(* IEC 61131-3 sources: elnaProjects/ElpcLogic/PomarKc7Unchanged/build_USO_ecl (part 7) *)

                                          StrAlg.inOpcCommandsDisabled:=FALSE;

  				cmd_for_Status := cmd;
  				source_for_Status := source;
  				command_error_for_Status := 0;
  	END_CASE;
  	resetCmdTimer(IN := false);
  	resetCmdTimerPriznak := TRUE;
  END_IF;
  lastCmd := cmd;

  resetCmdTimer(IN := resetCmdTimerPriznak, PT := T#5S);
  IF resetCmdTimer.Q THEN
  	resetCmdTimerPriznak := FALSE;
  	source_for_Status := 0;
  	cmd_for_Status := 0;
  	command_error_for_Status := 0;
  END_IF;

  StrAlg.Start:= puskOilSystem.startStatus
              OR nuOff.startStatus
              OR dPmgAi.startStatus
              OR dPmgDi.startStatus
              OR nuOn.startStatus
              OR noRezrv.startStatus
              OR BreakTest.startStatus
              OR testUnsuccessful.startStatus
              OR pnsOff.startStatus
              OR stopANU.startStatus
              OR nu1Off.startStatus
              OR nu2Off.startStatus;

  StrAlg.Error:=  puskOilSystem.errorStatus
              OR nuOff.errorStatus
              OR dPmgAi.errorStatus
              OR dPmgDi.errorStatus
              OR nuOn.errorStatus
              OR noRezrv.errorStatus
              OR BreakTest.errorStatus
              OR testUnsuccessful.errorStatus
              OR pnsOff.errorStatus
              OR stopANU.errorStatus
              OR nu1Off.errorStatus
              OR nu2Off.errorStatus;

  StrAlg.Top:=   puskOilSystem.topStatus
              OR nuOff.topStatus
              OR dPmgAi.topStatus
              OR dPmgDi.topStatus
              OR nuOn.topStatus
              OR noRezrv.topStatus
              OR BreakTest.topStatus
              OR testUnsuccessful.topStatus
              OR pnsOff.topStatus
              OR stopANU.topStatus
              OR nu1Off.topStatus
              OR nu2Off.topStatus;

  (*TODO: TYPE PROGRAM CODE HERE*)
  StrAlg.status :=  SHL(BYTE_TO_DWORD(source_for_Status), 29)
  			OR SHL(BYTE_TO_DWORD(cmd_for_Status), 26)
  			OR SHL(BYTE_TO_DWORD(command_error_for_Status), 23)
  			OR SHL(BOOL_TO_DWORD(StrAlg.OpcCommandsDisabled ), 21)
  			OR SHL(BOOL_TO_DWORD(StrAlg.hasError),4)
  			OR SHL(BOOL_TO_DWORD(StrAlg.CanRun),2)
  			OR SHL(BOOL_TO_DWORD(StrAlg.isEnded),1)
  			OR BOOL_TO_DWORD(StrAlg.isRuning);
END_FUNCTION_BLOCK

FUNCTION_BLOCK fb_ph_AIprotection
  VAR_IN_OUT
    StrAiP : struct_AiProtection;
  END_VAR
  VAR_INPUT
    act : TYPE_PhaseAlgoritmAction;
    PhaseNumber : UINT;
  END_VAR
  VAR_IN_OUT
    StrPh : struct_PhaseAlgoritm;
  END_VAR
  VAR
    CommandFault_Trig : R_TRIG;
    reset_Trig : R_TRIG;
    _statusDualInput : TYPE_statusDualInput;
  END_VAR

  IF StrPh.run AND NOT StrPh.start THEN
  	StrPh.start := TRUE;
  	StrPh.top := FALSE;
  	StrPh.error := FALSE;
            StrPh.run:=FALSE;

  	CASE act OF
  		(*PhaseAlgoritmAction.run*)    _run : runAiProtection(StrAiP); (*cmd_run*)
  		(*PhaseAlgoritmAction.reset*)_reset : resetAiProtection(StrAiP); (*cmd_reset*)
  	END_CASE;
  END_IF;

  IF StrPh.start AND NOT StrPh.top THEN
                      CommandFault_Trig(CLK := StrAiP.hasError);
                      IF CommandFault_Trig.Q THEN
  	          StrPh.error := TRUE;
                      END_IF;

  		CASE act OF
  		(*PhaseAlgoritmAction.run*)    _run:    StrPh.top:=StrAiP.isRunning;

  		(*PhaseAlgoritmAction.reset*) _reset:   StrPh.top := NOT StrAiP.isRunning;
  		END_CASE;

  END_IF;

  IF StrPh.top THEN
  StrPh.error := FALSE;
  END_IF;

  reset_Trig(CLK := StrPh.reset);
  IF reset_Trig.Q THEN
            StrPh.start := FALSE;
  	StrPh.error := FALSE;
  	StrPh.top := FALSE;
            StrPh.run:=FALSE;
            StrPh.reset:=FALSE;
  END_IF;

  StrPh.startStatus := SHL(BOOL_TO_DWORD(StrPh.start), PhaseNumber);
  StrPh.errorStatus := SHL(BOOL_TO_DWORD(StrPh.error), PhaseNumber);
  StrPh.topStatus := SHL(BOOL_TO_DWORD(StrPh.top), PhaseNumber);
END_FUNCTION_BLOCK

FUNCTION_BLOCK testPmsAlg
  VAR_IN_OUT
    StrAlg : struct_Alg;
    algContinue : struct_Question;
  END_VAR
  VAR
    pnsOn : struct_PhaseAlgoritm;
    PmsUp : struct_PhaseAlgoritm;
    runProtecrionAi : struct_PhaseAlgoritm;
    pnsOff : struct_PhaseAlgoritm;
    BreakTest : struct_PhaseAlgoritm;
    LowOilPS : struct_PhaseAlgoritm;
    LowOilAS : struct_PhaseAlgoritm;
    testUnsuccessful : struct_PhaseAlgoritm;
    fb_pnsOn : fb_ph_Switch;
    fb_PmsUp : fb_ph_WaitAnalogValue;
    fb_algContinue : fb_Question;
    fb_runProtecrionAi : fb_ph_AIprotection;
    fb_pnsOff : fb_ph_Switch;
    fb_BreakTest : fb_ph_Timer;
    fb_LowOilPS : fb_ph_CustomPhase;
    fb_LowOilAS : fb_ph_CustomPhase;
    fb_testUnsuccessful : fb_ph_CustomPhase;
    _sunpackerCommand : fb_sunpackerCommand;
    _DualStateImAction : TYPE_DualStateImAction;
    _Answers : TYPE_Answers;
    _statusDualInput : TYPE_statusDualInput;
    _StatusAi : TYPE_StatusAi;
    _PhaseAlgoritmAction : TYPE_PhaseAlgoritmAction;
    source : BYTE;
    cmd : BYTE;
    lastCmd : BYTE;
    source_for_Status : BYTE;
    cmd_for_Status : BYTE;
    command_error_for_Status : BYTE;
    resetCmdTimer : TON;
    resetCmdTimerPriznak : BOOL;
    onInit : BOOL;
    _resetQuestion : BOOL;
    waitReset : TON;
  END_VAR
  VAR_EXTERNAL
    IM : ImConfig;
    algoritms : AlgoritmsConfig;
    ai : AiConfig;
    AlgTimers : struct_AlgTimers;
    ModeGpa : TYPE_ModeGpa;
    algManager : struct_AlgoritmsManager;
    protections : ProtectionsConfig;
  END_VAR

  IF NOT onInit THEN

                     fb_pnsOn(phaseNumber:=0, act:=_on);
          algContinue.AnswerVariants:=_Answers.ANS_YES;
                     fb_PmsUp(phaseNumber:=1);
           fb_runProtecrionAi(phaseNumber:=3, act:=_run);
                    fb_pnsOff(phaseNumber:=4, act:=_off);
                 fb_BreakTest(phaseNumber:=5, delay:=T#120S);
                  fb_LowOilPS(phaseNumber:=6);
                  fb_LowOilAS(phaseNumber:=7);
          fb_testUnsuccessful(phaseNumber:=8);

  onInit:=TRUE;
  END_IF;

              fb_pnsOn(StrPh:=pnsOn, Im:=IM.pns);
        fb_algContinue(StrQ:=algContinue);
              fb_PmsUp(StrPh:=PmsUp, ai:=ai.P_masla_smazki_nizkoe, more:=ai.P_masla_smazki_nizkoe.LW);
    fb_runProtecrionAi(StrPh:=runProtecrionAi, StrAiP:=protections.P_masla_smazki_nizkoe_LA);
             fb_pnsOff(StrPh:=pnsOff, Im:=IM.pns);
          fb_BreakTest(StrPh:=BreakTest, timer:=AlgTimers.testPms_BreakTest);
           fb_LowOilPS(StrPh:=LowOilPS);
           fb_LowOilAS(StrPh:=LowOilAS);
   fb_testUnsuccessful(StrPh:=testUnsuccessful);

  StrAlg.CanRun := StrAlg.inCanRun;
  StrAlg.OpcCommandsDisabled := StrAlg.inOpcCommandsDisabled;

  IF StrAlg.isRuning THEN

      StrAlg.hasError := pnsOn.error OR pnsOff.error OR testUnsuccessful.error;

      IF pnsOn.top THEN
           runPhase(PmsUp);
      END_IF;

      IF PmsUp.top THEN
           runPhase(runProtecrionAi);
      END_IF;

      IF runProtecrionAi.top THEN
           IM.SingleSignals.P_oil_low.Disabled_Sig:=FALSE;
           ai.P_masla_smazki_nizkoe.Disabled_LA:=FALSE;
           ai.P_masla_smazki_nizkoe.Disabled_LW:=FALSE;
           ai.P_masla_smazki_srednee_posle_nasosov.Disabled_LW:=FALSE;
               IF NOT _resetQuestion THEN
                   askQuestion(algContinue);
                   _resetQuestion:=TRUE;
               END_IF;
      END_IF;

      IF algContinue.answer = _Answers.ANS_YES THEN

          runPhase(BreakTest);
          runPhase(pnsOff);
          runPhase(LowOilPS);
          runPhase(LowOilAS);
          resetQuestion(algContinue);

      END_IF;

      IF 	LowOilPS.start AND NOT LowOilPS.top THEN
  	LowOilPS.top:= ai.P_masla_smazki_nizkoe.interval = _statusAi.LW;
      END_IF;
      IF 	LowOilAS.start AND NOT LowOilAS.top THEN
  	LowOilAS.top:= ai.P_masla_smazki_nizkoe.interval = _statusAi.LA;
      END_IF;

      IF LowOilPS.top AND LowOilAS.top THEN
            resetPhase(BreakTest);
            waitReset(IN:=TRUE, PT:= T#3S);
      END_IF;

      IF BreakTest.top AND StrAlg.isEnded THEN
  	testUnsuccessful.error:=TRUE;
      END_IF;

      IF waitReset.Q THEN
          algManager.nMode:=ModeGpa.MODE_STOP;
          resetIfRunning(StrAlg);
      END_IF;

      StrAlg.isEnded:= LowOilPS.top AND LowOilAS.top;

  END_IF;

  StrAlg.CanRun := StrAlg.inCanRun;
  StrAlg.OpcCommandsDisabled := StrAlg.inOpcCommandsDisabled;

  (* ---- Если управление с ВУ заблокировано, то  передаем команду из алгоритма ---- *)
  IF StrAlg.inOpcCommandsDisabled THEN
  	StrAlg.inCommand := StrAlg.inCommand_Alg;
  ELSE (* иначе передаем команду с АРМа*)
  	StrAlg.inCommand := StrAlg.inCommand_ARM;
  END_IF;

  _sunpackerCommand(command := StrAlg.inCommand);
  	source := _sunpackerCommand.source;
  	cmd := _sunpackerCommand.cmd;

  IF cmd <> 0 AND lastCmd <> cmd AND (((NOT StrAlg.opcCommandsDisabled) AND source > 0) OR source = 0) then
  	CASE BYTE_TO_INT(cmd) OF
  		(*cmdRun*) 1: 	IF (StrAlg.CanRun) THEN
  					StrAlg.isRuning := TRUE;
  					StrAlg.isEnded := FALSE;
  					StrAlg.hasError := FALSE;
  					(*****************       OnRun       *****************)

                                                    algManager.nMode:=ModeGpa.MODE_TESTPMS;
                                                    resetAndDisable(alg:=algoritms.ppu);
                                                    runPhase(pnsOn);

  					cmd_for_Status := cmd;
  					source_for_Status := source;
  					command_error_for_Status := 0;
  				ELSE
  					StrAlg.isRuning := FALSE;
  					StrAlg.isEnded := FALSE;
  					StrAlg.hasError 	:= FALSE;

  					cmd_for_Status := 0;
  					source_for_Status := source;
  					command_error_for_Status := cmd;
  				END_IF;
  		(*cmdReset*) 2: 	StrAlg.isRuning := FALSE;
  				StrAlg.isEnded := FALSE;
  				StrAlg.hasError 	:= FALSE;

                                           (*****************       OnReset       *****************)
                                          waitReset(IN:=FALSE);
                                          _resetQuestion:=FALSE;
                                          ai.P_masla_smazki_nizkoe.Disabled_LA:=TRUE;
                                          ai.P_masla_smazki_nizkoe.Disabled_LW:=TRUE;
                                          ai.P_masla_smazki_srednee_posle_nasosov.Disabled_LW:=TRUE;
                                          IM.SingleSignals.P_oil_low.Disabled_Sig:=TRUE;
                                          resetAiProtection(protections.P_masla_smazki_nizkoe_LA);

                                          resetPhase(pnsOn);
                                          resetPhase(PmsUp);
                                          resetPhase(runProtecrionAi);
                                          resetPhase(pnsOff);
                                          resetPhase(BreakTest);
                                          resetPhase(LowOilPS);
                                          resetPhase(LowOilAS);
                                          resetPhase(testUnsuccessful);

                                          resetQuestion(algContinue);

                                          StrAlg.inOpcCommandsDisabled:=FALSE;

  				cmd_for_Status := cmd;
  				source_for_Status := source;
  				command_error_for_Status := 0;
  	END_CASE;
  	resetCmdTimer(IN := false);
  	resetCmdTimerPriznak := TRUE;
  END_IF;
  lastCmd := cmd;

  resetCmdTimer(IN := resetCmdTimerPriznak, PT := T#5S);
  IF resetCmdTimer.Q THEN
  	resetCmdTimerPriznak := FALSE;
  	source_for_Status := 0;
  	cmd_for_Status := 0;
  	command_error_for_Status := 0;
  END_IF;

  StrAlg.Start:= pnsOn.startStatus
              OR PmsUp.startStatus
              OR runProtecrionAi.startStatus
              OR pnsOff.startStatus
              OR BreakTest.startStatus
              OR LowOilPS.startStatus
              OR LowOilAS.startStatus
              OR testUnsuccessful.startStatus;

  StrAlg.Error:= pnsOn.errorStatus
              OR PmsUp.errorStatus
              OR runProtecrionAi.errorStatus
              OR pnsOff.errorStatus
              OR BreakTest.errorStatus
              OR LowOilPS.errorStatus
              OR LowOilAS.errorStatus
              OR testUnsuccessful.errorStatus;

  StrAlg.Top:=   pnsOn.topStatus
              OR PmsUp.topStatus
              OR runProtecrionAi.topStatus
              OR pnsOff.topStatus
              OR BreakTest.topStatus
              OR LowOilPS.topStatus
              OR LowOilAS.topStatus
              OR testUnsuccessful.topStatus;

  (*TODO: TYPE PROGRAM CODE HERE*)
  StrAlg.status :=  SHL(BYTE_TO_DWORD(source_for_Status), 29)
  			OR SHL(BYTE_TO_DWORD(cmd_for_Status), 26)
  			OR SHL(BYTE_TO_DWORD(command_error_for_Status), 23)
  			OR SHL(BOOL_TO_DWORD(StrAlg.OpcCommandsDisabled ), 21)
  			OR SHL(BOOL_TO_DWORD(StrAlg.hasError),4)
  			OR SHL(BOOL_TO_DWORD(StrAlg.CanRun),2)
  			OR SHL(BOOL_TO_DWORD(StrAlg.isEnded),1)
  			OR BOOL_TO_DWORD(StrAlg.isRuning);
END_FUNCTION_BLOCK

FUNCTION_BLOCK ApuskAlg
  VAR_IN_OUT
    StrAlg : struct_Alg;
  END_VAR
  VAR
    runOilsystem : struct_PhaseAlgoritm;
    runEngine : struct_PhaseAlgoritm;
    filling : struct_PhaseAlgoritm;
    fb_runOilsystem : fb_ph_algoritm;
    fb_runEngine : fb_ph_algoritm;
    fb_filling : fb_ph_algoritm;
    _sunpackerCommand : fb_sunpackerCommand;
    _PhaseAlgoritmAction : TYPE_PhaseAlgoritmAction;
    _statusDualInput : TYPE_statusDualInput;
    source : BYTE;
    cmd : BYTE;
    lastCmd : BYTE;
    source_for_Status : BYTE;
    cmd_for_Status : BYTE;
    command_error_for_Status : BYTE;
    resetCmdTimer : TON;
    resetCmdTimerPriznak : BOOL;
    onInit : BOOL;
    waitReset : TON;
  END_VAR
  VAR_EXTERNAL
    algoritms : AlgoritmsConfig;
    ModeGpa : TYPE_ModeGpa;
    algManager : struct_AlgoritmsManager;
    IM : ImConfig;
  END_VAR

  IF NOT onInit THEN

           fb_runOilsystem(phaseNumber:=0, act:=_run, waitCompletion:=TRUE);
              fb_runEngine(phaseNumber:=1, act:=_run, waitCompletion:=TRUE);
                fb_filling(phaseNumber:=2, act:=_run, waitCompletion:=TRUE);

  onInit:=TRUE;
  END_IF;

           fb_runOilsystem(StrPh:=runOilsystem, alg:=algoritms.puskOilSystem);
              fb_runEngine(StrPh:=runEngine, alg:=algoritms.engineRun);
                fb_filling(StrPh:=filling, alg:=algoritms.filling);

  StrAlg.CanRun := StrAlg.inCanRun;
  StrAlg.OpcCommandsDisabled := StrAlg.inOpcCommandsDisabled;

  IF StrAlg.isRuning THEN

      StrAlg.hasError := runOilsystem.error OR runEngine.error OR filling.error;

      IF runOilsystem.top THEN
           runPhase(runEngine);
      END_IF;

      IF runEngine.top THEN
           runPhase(filling);
      END_IF;

      IF filling.top THEN
            waitReset(IN:=TRUE, PT:= T#2S);
      END_IF;

      IF waitReset.Q THEN

          IF Im.kran6.onStatus = _statusDualInput.STATUS_On THEN
  	algManager.nMode:= ModeGpa.MODE_WORK_Ring;
          END_IF;
          IF Im.kran6.onStatus = _statusDualInput.STATUS_Off THEN
  	algManager.nMode:= ModeGpa.MODE_WORK_Line;
          END_IF;

          resetIfRunning(StrAlg);
      END_IF;

      StrAlg.isEnded:= filling.top;

  END_IF;

  StrAlg.CanRun := StrAlg.inCanRun;
  StrAlg.OpcCommandsDisabled := StrAlg.inOpcCommandsDisabled;

  (* ---- Если управление с ВУ заблокировано, то  передаем команду из алгоритма ---- *)
  IF StrAlg.inOpcCommandsDisabled THEN
  	StrAlg.inCommand := StrAlg.inCommand_Alg;
  ELSE (* иначе передаем команду с АРМа*)
  	StrAlg.inCommand := StrAlg.inCommand_ARM;
  END_IF;

  _sunpackerCommand(command := StrAlg.inCommand);
  	source := _sunpackerCommand.source;
  	cmd := _sunpackerCommand.cmd;

  IF cmd <> 0 AND lastCmd <> cmd AND (((NOT StrAlg.opcCommandsDisabled) AND source > 0) OR source = 0) then
  	CASE BYTE_TO_INT(cmd) OF
  		(*cmdRun*) 1: 	IF (StrAlg.CanRun) THEN
  					StrAlg.isRuning := TRUE;
  					StrAlg.isEnded := FALSE;
  					StrAlg.hasError := FALSE;
  					(*****************       OnRun       *****************)

                                                    algoritms.puskOilSystem.inCanRun:= TRUE	;
                                                    algoritms.filling.inCanRun:= TRUE	;
                                                    algoritms.engineRun.inCanRun:= TRUE	;

                                                    algManager.nMode:=ModeGpa.MODE_APUSK;
                                                    impulseSO(Im.SingleOutputs.VzvodBREO);
                                                    runPhase(runOilsystem);

  					cmd_for_Status := cmd;
  					source_for_Status := source;
  					command_error_for_Status := 0;
  				ELSE
  					StrAlg.isRuning := FALSE;
  					StrAlg.isEnded := FALSE;
  					StrAlg.hasError 	:= FALSE;

  					cmd_for_Status := 0;
  					source_for_Status := source;
  					command_error_for_Status := cmd;
  				END_IF;
  		(*cmdReset*) 2: 	StrAlg.isRuning := FALSE;
  				StrAlg.isEnded := FALSE;
  				StrAlg.hasError 	:= FALSE;

                                           (*****************       OnReset       *****************)
                                          waitReset(IN:=FALSE);
                                          StrAlg.inCanRun:=FALSE;

                                          resetPhase(runOilsystem);
                                          resetPhase(runEngine);
                                          resetPhase(filling);

                                          StrAlg.inOpcCommandsDisabled:=FALSE;

  				cmd_for_Status := cmd;
  				source_for_Status := source;
  				command_error_for_Status := 0;
  	END_CASE;
  	resetCmdTimer(IN := false);
  	resetCmdTimerPriznak := TRUE;
  END_IF;
  lastCmd := cmd;

  resetCmdTimer(IN := resetCmdTimerPriznak, PT := T#5S);
  IF resetCmdTimer.Q THEN
  	resetCmdTimerPriznak := FALSE;
  	source_for_Status := 0;
  	cmd_for_Status := 0;
  	command_error_for_Status := 0;
  END_IF;

  StrAlg.Start:= runOilsystem.startStatus
              OR runEngine.startStatus
              OR filling.startStatus;

  StrAlg.Error:= runOilsystem.errorStatus
              OR runEngine.errorStatus
              OR filling.errorStatus;

  StrAlg.Top:=   runOilsystem.topStatus
              OR runEngine.topStatus
              OR filling.topStatus;

  (*TODO: TYPE PROGRAM CODE HERE*)
  StrAlg.status :=  SHL(BYTE_TO_DWORD(source_for_Status), 29)
  			OR SHL(BYTE_TO_DWORD(cmd_for_Status), 26)
  			OR SHL(BYTE_TO_DWORD(command_error_for_Status), 23)
  			OR SHL(BOOL_TO_DWORD(StrAlg.OpcCommandsDisabled ), 21)
  			OR SHL(BOOL_TO_DWORD(StrAlg.hasError),4)
  			OR SHL(BOOL_TO_DWORD(StrAlg.CanRun),2)
  			OR SHL(BOOL_TO_DWORD(StrAlg.isEnded),1)
  			OR BOOL_TO_DWORD(StrAlg.isRuning);
END_FUNCTION_BLOCK

FUNCTION_BLOCK SemiAutoPuskAlg
  VAR_IN_OUT
    StrAlg : struct_Alg;
  END_VAR
  VAR
    runOilsystem : struct_PhaseAlgoritm;
    runEngine : struct_PhaseAlgoritm;
    filling : struct_PhaseAlgoritm;
  END_VAR
  VAR_IN_OUT
    cmdRun1ph : struct_Question;
    cmdRun2ph : struct_Question;
    cmdRun3ph : struct_Question;
  END_VAR
  VAR
    fb_runOilsystem : fb_ph_algoritm;
    fb_runEngine : fb_ph_algoritm;
    fb_filling : fb_ph_algoritm;
    fb_cmdRun1ph : fb_Question;
    fb_cmdRun2ph : fb_Question;
    fb_cmdRun3ph : fb_Question;
    _sunpackerCommand : fb_sunpackerCommand;
    _PhaseAlgoritmAction : TYPE_PhaseAlgoritmAction;
    _statusDualInput : TYPE_statusDualInput;
    _Answers : TYPE_Answers;
    source : BYTE;
    cmd : BYTE;
    lastCmd : BYTE;
    source_for_Status : BYTE;
    cmd_for_Status : BYTE;
    command_error_for_Status : BYTE;
    resetCmdTimer : TON;
    resetCmdTimerPriznak : BOOL;
    onInit : BOOL;
    waitReset : TON;
  END_VAR
  VAR_EXTERNAL
    algoritms : AlgoritmsConfig;
    ModeGpa : TYPE_ModeGpa;
    algManager : struct_AlgoritmsManager;
    IM : ImConfig;
  END_VAR

  IF NOT onInit THEN
                 cmdRun1ph.AnswerVariants:=_Answers.ANS_YES;
           fb_runOilsystem(phaseNumber:=0, act:=_run, waitCompletion:=TRUE);
                 cmdRun2ph.AnswerVariants:=_Answers.ANS_YES;
              fb_runEngine(phaseNumber:=1, act:=_run, waitCompletion:=TRUE);
                 cmdRun3ph.AnswerVariants:=_Answers.ANS_YES;
                fb_filling(phaseNumber:=2, act:=_run, waitCompletion:=TRUE);

  onInit:=TRUE;
  END_IF;
              fb_cmdRun1ph(StrQ:=cmdRun1ph);
           fb_runOilsystem(StrPh:=runOilsystem, alg:=algoritms.puskOilSystem);
              fb_cmdRun2ph(StrQ:=cmdRun2ph);
              fb_runEngine(StrPh:=runEngine, alg:=algoritms.engineRun);
              fb_cmdRun3ph(StrQ:=cmdRun3ph);
                fb_filling(StrPh:=filling, alg:=algoritms.filling);

  StrAlg.CanRun := StrAlg.inCanRun;
  StrAlg.OpcCommandsDisabled := StrAlg.inOpcCommandsDisabled;

  IF StrAlg.isRuning THEN

      StrAlg.hasError := runOilsystem.error OR runEngine.error OR filling.error;

      IF cmdRun1ph.answer = _Answers.ANS_YES THEN
  	runPhase(runOilsystem);
            resetQuestion(cmdRun1ph);
      END_IF;

      IF runOilsystem.top AND NOT runEngine.start THEN
           askQuestion(cmdRun2ph);
      END_IF;

      IF cmdRun2ph.answer = _Answers.ANS_YES THEN
           runPhase(runEngine);
           resetQuestion(cmdRun2ph);
      END_IF;

      IF runEngine.top AND NOT filling.start THEN
           askQuestion(cmdRun3ph);
      END_IF;

      IF cmdRun3ph.answer = _Answers.ANS_YES THEN
           runPhase(filling);
           resetQuestion(cmdRun3ph);
      END_IF;

      IF filling.top THEN
            waitReset(IN:=TRUE, PT:= T#2S);
      END_IF;

      IF waitReset.Q THEN

          IF Im.kran6.onStatus = _statusDualInput.STATUS_On THEN
  	algManager.nMode:= ModeGpa.MODE_WORK_Ring;
          END_IF;
          IF Im.kran6.onStatus = _statusDualInput.STATUS_Off THEN
  	algManager.nMode:= ModeGpa.MODE_WORK_Line;
          END_IF;

          resetIfRunning(StrAlg);
      END_IF;

      StrAlg.isEnded:= filling.top;

  END_IF;

  StrAlg.CanRun := StrAlg.inCanRun;
  StrAlg.OpcCommandsDisabled := StrAlg.inOpcCommandsDisabled;

  (* ---- Если управление с ВУ заблокировано, то  передаем команду из алгоритма ---- *)
  IF StrAlg.inOpcCommandsDisabled THEN
  	StrAlg.inCommand := StrAlg.inCommand_Alg;
  ELSE (* иначе передаем команду с АРМа*)
  	StrAlg.inCommand := StrAlg.inCommand_ARM;
  END_IF;

  _sunpackerCommand(command := StrAlg.inCommand);
  	source := _sunpackerCommand.source;
  	cmd := _sunpackerCommand.cmd;

  IF cmd <> 0 AND lastCmd <> cmd AND (((NOT StrAlg.opcCommandsDisabled) AND source > 0) OR source = 0) then
  	CASE BYTE_TO_INT(cmd) OF
  		(*cmdRun*) 1: 	IF (StrAlg.CanRun) THEN
  					StrAlg.isRuning := TRUE;
  					StrAlg.isEnded := FALSE;
  					StrAlg.hasError := FALSE;
  					(*****************       OnRun       *****************)

                                                    algoritms.puskOilSystem.inCanRun:= TRUE	;
                                                    algoritms.filling.inCanRun:= TRUE	;
                                                    algoritms.engineRun.inCanRun:= TRUE	;

                                                    algManager.nMode:=ModeGpa.MODE_MPUSK;
                                                    impulseSO(Im.SingleOutputs.VzvodBREO);
                                                    askQuestion(cmdRun1ph);

  					cmd_for_Status := cmd;
  					source_for_Status := source;
  					command_error_for_Status := 0;
  				ELSE
  					StrAlg.isRuning := FALSE;
  					StrAlg.isEnded := FALSE;
  					StrAlg.hasError 	:= FALSE;

  					cmd_for_Status := 0;
  					source_for_Status := source;
  					command_error_for_Status := cmd;
  				END_IF;
  		(*cmdReset*) 2: 	StrAlg.isRuning := FALSE;
  				StrAlg.isEnded := FALSE;
  				StrAlg.hasError 	:= FALSE;

                                           (*****************       OnReset       *****************)
                                          waitReset(IN:=FALSE);
                                          StrAlg.inCanRun:=FALSE;

                                          resetPhase(runOilsystem);
                                          resetPhase(runEngine);
                                          resetPhase(filling);

                                          resetQuestion(cmdRun1ph);
                                          resetQuestion(cmdRun2ph);
                                          resetQuestion(cmdRun3ph);

                                          StrAlg.inOpcCommandsDisabled:=FALSE;

  				cmd_for_Status := cmd;
  				source_for_Status := source;
  				command_error_for_Status := 0;
  	END_CASE;
  	resetCmdTimer(IN := false);
  	resetCmdTimerPriznak := TRUE;
  END_IF;
  lastCmd := cmd;

  resetCmdTimer(IN := resetCmdTimerPriznak, PT := T#5S);
  IF resetCmdTimer.Q THEN
  	resetCmdTimerPriznak := FALSE;
  	source_for_Status := 0;
  	cmd_for_Status := 0;
  	command_error_for_Status := 0;
  END_IF;

  StrAlg.Start:= runOilsystem.startStatus
              OR runEngine.startStatus
              OR filling.startStatus;

  StrAlg.Error:= runOilsystem.errorStatus
              OR runEngine.errorStatus
              OR filling.errorStatus;

  StrAlg.Top:=   runOilsystem.topStatus
              OR runEngine.topStatus
              OR filling.topStatus;

  (*TODO: TYPE PROGRAM CODE HERE*)
  StrAlg.status :=  SHL(BYTE_TO_DWORD(source_for_Status), 29)
  			OR SHL(BYTE_TO_DWORD(cmd_for_Status), 26)
  			OR SHL(BYTE_TO_DWORD(command_error_for_Status), 23)
  			OR SHL(BOOL_TO_DWORD(StrAlg.OpcCommandsDisabled ), 21)
  			OR SHL(BOOL_TO_DWORD(StrAlg.hasError),4)
  			OR SHL(BOOL_TO_DWORD(StrAlg.CanRun),2)
  			OR SHL(BOOL_TO_DWORD(StrAlg.isEnded),1)
  			OR BOOL_TO_DWORD(StrAlg.isRuning);
END_FUNCTION_BLOCK

FUNCTION_BLOCK proc_algoritms
  VAR
    fb_RemontAlg : RemontAlg;
    fb_TestProtectionAlg : TestProtectionAlg;
    fb_TestImAlg : TestImAlg;
    fb_AutoTen : fb_AutoTenAlg;
    fb_AutoPns : fb_AutoPnsAlg;
    fb_AutoAvom : fb_AutoAvomAlg;
    fb_vibegPNS : fb_vibegPNSAlg;
    fb_AutoNU : fb_AutoNUAlg;
    fb_puskOilSystem : fb_puskOilSystemAlg;
    fb_AntiPompag : fb_AntiPompagAlg;
    fb_NOAlg : NOAlg;
    fb_AOAlg : AOAlg;
    fb_ppuALG : ppuAlg;
    fb_fillingAlg : fillingAlg;
    fb_engineRunAlg : engineRunAlg;
    fb_puskKalg : puskKalg;
    fb_puskValg : puskValg;
    fb_testdPmgAlg : testdPmgAlg;
    fb_testPmsAlg : testPmsAlg;
    fb_ApuskAlg : ApuskAlg;
    fb_SemiAutoPuskAlg : SemiAutoPuskAlg;
  END_VAR
  VAR_EXTERNAL
    algoritms : AlgoritmsConfig;
    AlgQuestions : AlgoritmsQuestions;
    ai : AiConfig;
    IM : ImConfig;
    AlgTimers : struct_AlgTimers;
  END_VAR

  fb_RemontAlg(StrAlg:=algoritms.Remont);

  fb_TestProtectionAlg(StrAlg:=algoritms.TestProtection);

  fb_TestImAlg(StrAlg:=algoritms.testIm);

  fb_AutoTen(StrAlg:= algoritms.AutoTen,
  T_masla:= ai.T_masla_v_maslobake,
  Uroven_masla:= ai.Uroven_masla_v_maslobake,
  offTemperature:= Im.AutoTen_offTemperature,
  TEN:= Im.Ten,
  PNS:= Im.pns);

  fb_AutoPns(StrAlg:= algoritms.AutoPns,
  Poil:= ai.P_masla_smazki_nizkoe,
  Ust_Run:= Im.AutoPns_UstRun,
  Ust_Stop:= Im.AutoPns_UstStop,
  Nasos:= Im.pns,
  diPlow:= Im.SingleSignals.P_oil_low);

  fb_AutoAvom(StrAlg:= algoritms.AutoAvom,
  im1:= Im.v1_Avom,
  im2:= Im.v2_Avom,
  on1Temperature:= Im.AutoAvom_onTemp1,
  on2Temperature:= Im.AutoAvom_onTemp2,
  hystereses:= Im.AutoAvom_hysteresis,
  ai:= ai.T_masla_posle_AVOM);

  fb_vibegPNS(StrAlg:=algoritms.vibegPNS,
  algContinue:=AlgQuestions.vibegPNS_algContinue
  );

  fb_AutoNU(StrAlg:=algoritms.autoNu,
  nu1:=Im.nu1,
  nu2:=Im.nu2,
  Ust_Swap:= Im.AutoNU_Ust_Swap,
  mainNU:= Im.AutoNU_mainNU,
  dPoil:=ai.dPmaslo_gaz,
  Lowdp_di:=Im.SingleSignals.dP_oilgaz_low
  );

  fb_puskOilSystem(StrAlg:=algoritms.puskOilSystem);

  fb_AntiPompag(StrAlg:=algoritms.AntiPompag,
  Rashod:= ai.Rashod,
  Zapas:= ai.Zapas,
  P_gasIn:=ai.P_gaza_na_vkhode_nagnetatelia,
  T_gasIn:=ai.T_gaz_in_nagnetatelia,
  dP_konf:=ai.dP_gaza_na_konfuzore_nagnetatelia,
  Kran6:= im.Kran6,
  UgolVNA:= im.AntiPompag_UgolVNA,
  K:=im.AntiPompag_K,
  A:=im.AntiPompag_A,
  y0:=im.AntiPompag_y0);

  fb_NOAlg(StrAlg:=algoritms.no);

  fb_AOAlg(StrAlg:=algoritms.ao);

  fb_ppuAlg(StrAlg:=algoritms.ppu);

  fb_fillingAlg(StrAlg:=algoritms.filling);

  fb_engineRunAlg(StrAlg:=algoritms.engineRun);

  fb_puskKalg(StrAlg:=algoritms.puskK,
  questionFilling:=AlgQuestions.puskK_questionFilling,
   questionUnload:=AlgQuestions.puskK_questionUnload
  );

  fb_puskValg(StrAlg:=algoritms.puskV,
   questionEngine:=AlgQuestions.puskV_questionEngine,
    questionMVoff:=AlgQuestions.puskV_questionMVoff
  );

  fb_testdPmgAlg(StrAlg:=algoritms.testdPmg,
   algContinue:=AlgQuestions.testdPmg_algContinue
  );

  fb_testPmsAlg(StrAlg:=algoritms.testPms,
   algContinue:=AlgQuestions.testPms_algContinue
  );

  fb_ApuskAlg(StrAlg:=algoritms.Apusk);

  fb_SemiAutoPuskAlg(StrAlg:=algoritms.SemiAutoPusk,
   cmdRun1ph:=AlgQuestions.SemiAutoPusk_cmdRun1ph,
   cmdRun2ph:=AlgQuestions.SemiAutoPusk_cmdRun2ph,
   cmdRun3ph:=AlgQuestions.SemiAutoPusk_cmdRun3ph
  );
END_FUNCTION_BLOCK

FUNCTION anyProtectionSignaling : BOOL
  VAR_INPUT
    protections : ProtectionsConfig;
  END_VAR

  anyProtectionSignaling:=
  protections.T_perednego_opornogo_podshipnika_dvigatelia_t1_HA.Signaling OR
  protections.T_zadnego_opornogo_podshipnika_dvigatelia_t2_HA.Signaling OR
  protections.T_podshipnika_reduktora_t1_HA.Signaling OR
  protections.T_podshipnika_reduktora_t2_HA.Signaling OR
  protections.T_podshipnika_reduktora_t3_HA.Signaling OR
  protections.T_podshipnika_reduktora_t4_HA.Signaling OR
  protections.T_opornogo_podshipnika_nagnetatelia_t1_HA.Signaling OR
  protections.T_opornogo_podshipnika_nagnetatelia_t2_HA.Signaling OR
  protections.T_opornogo_podshipnika_nagnetatelia_t3_HA.Signaling OR
  protections.T_opornoupornogo_podshipnika_nagnetatelia_t4_HA.Signaling OR
  protections.T_gaza_na_vykhode_nagnetatelia_HA.Signaling OR
  protections.dP_maslogaz_LA.Signaling OR
  protections.P_masla_smazki_nizkoe_LA.Signaling OR
  protections.Vibratciia_STD_t1_HA.Signaling OR
  protections.Vibratciia_STD_t2_HA.Signaling OR
  protections.Vibratciia_rotora_nagnetatelia_t1_HA.Signaling OR
  protections.Vibratciia_rotora_nagnetatelia_t2_HA.Signaling OR
  protections.Vibratciia_rotora_nagnetatelia_t3_HA.Signaling OR
  protections.Vibratciia_rotora_nagnetatelia_t4_HA.Signaling OR
  protections.Osevoi_sdvig_rotora_nagnetatelia_HA.Signaling OR
  protections.Uroven_masla_v_maslobake_LA.Signaling OR
  protections.OsevojSdvigPravyjDi.Signaling OR
  protections.OsevojSdvigLevyjDi.Signaling OR
  protections.dP_masloGaz_LowDI.Signaling OR
  protections.DavlenieMaslaSmazkiDi.Signaling OR
  protections.mvOff.Signaling OR
  protections.NeispravnostVozbuzhdenijaDi.Signaling OR
  protections.AO_KC.Signaling OR
  protections.AO_PRU.Signaling OR
  protections.AO_SHU.Signaling OR
  protections.Srab_BEAO.Signaling OR
  protections.EAO_PRU.Signaling OR
  protections.BEAO_knSHU.Signaling OR
  protections.Kran1sdvig.Signaling OR
  protections.Kran2sdvig.Signaling;
END_FUNCTION

FUNCTION anyAnalogsPs : BOOL
  VAR_INPUT
    ai : AiConfig;
  END_VAR
  VAR
    statusAi : TYPE_StatusAi;
  END_VAR

  anyAnalogsPs:=
  ai.T_masla_v_maslobake.interval= statusAi.HW OR
  ai.T_masla_v_maslobake.interval= statusAi.LW OR
  ai.T_perednego_opornogo_podshipnika_dvigatelia_t1.interval= statusAi.HW OR
  ai.T_zadnego_opornogo_podshipnika_dvigatelia_t2.interval= statusAi.HW OR
  ai.T_podshipnika_reduktora_t1.interval= statusAi.HW OR
  ai.T_podshipnika_reduktora_t2.interval= statusAi.HW OR
  ai.T_podshipnika_reduktora_t3.interval= statusAi.HW OR
  ai.T_podshipnika_reduktora_t4.interval= statusAi.HW OR
  ai.T_opornogo_podshipnika_nagnetatelia_t1.interval= statusAi.HW OR
  ai.T_opornogo_podshipnika_nagnetatelia_t2.interval= statusAi.HW OR
  ai.T_opornogo_podshipnika_nagnetatelia_t3.interval= statusAi.HW OR
  ai.T_oporno_upornogo_podshipnika_nagnetatelia_t4.interval= statusAi.HW OR
  ai.T_gaz_out_nagnetatelia.interval= statusAi.HW OR
  ai.dPmaslo_gaz.interval= statusAi.LW OR
  ai.P_masla_smazki_nizkoe.interval= statusAi.LW OR
  ai.P_masla_smazki_srednee_posle_nasosov.interval= statusAi.LW OR
  ai.Vibratciia_STD_t1.interval= statusAi.HW OR
  ai.Vibratciia_STD_t2.interval= statusAi.HW OR
  ai.Vibratciia_rotora_nagnetatelia_t1.interval= statusAi.HW OR
  ai.Vibratciia_rotora_nagnetatelia_t2.interval= statusAi.HW OR
  ai.Vibratciia_rotora_nagnetatelia_t3.interval= statusAi.HW OR
  ai.Vibratciia_rotora_nagnetatelia_t4.interval= statusAi.HW OR
  ai.Osevoi_sdvig_rotora_nagnetatelia.interval= statusAi.HW OR
  ai.Osevoi_sdvig_rotora_nagnetatelia.interval= statusAi.LW OR
  ai.Uroven_masla_v_maslobake.interval= statusAi.HW OR
  ai.Uroven_masla_v_maslobake.interval= statusAi.LW OR
  ai.T_vnytri_shkafa.interval= statusAi.HW OR
  ai.T_vnytri_shkafa.interval= statusAi.LW OR
  ai.VoltageSHU_osnovnoi_vvod.interval= statusAi.HW OR
  ai.VoltageSHU_osnovnoi_vvod.interval= statusAi.LW OR
  ai.VoltageSHU_rezervnyi_vvod.interval= statusAi.HW OR
  ai.VoltageSHU_rezervnyi_vvod.interval= statusAi.LW;
END_FUNCTION

FUNCTION anyDiscretPS : BOOL
  VAR_INPUT
    im : ImConfig;
  END_VAR

  anyDiscretPS:=
      Im.SingleSignals.KZ_10kv.Q                     OR
      Im.SingleSignals.Vozb_ProboiVentila.Q	 OR
      Im.SingleSignals.Vozb_AsinchHod.Q	           OR
      Im.SingleSignals.NS_ForsingVozbugdenia.Q       OR
      Im.SingleSignals.Vozb_AutoUprVozbuditela_off.Q OR
      Im.SingleSignals.Vozb_KontaktorON.Q;
END_FUNCTION

FUNCTION UnBlockAllProtections : BOOL
  VAR_IN_OUT
    protections : ProtectionsConfig;
  END_VAR

  protections.T_perednego_opornogo_podshipnika_dvigatelia_t1_HA.inOpcCommandsDisabled:=FALSE;
  protections.T_zadnego_opornogo_podshipnika_dvigatelia_t2_HA.inOpcCommandsDisabled:=FALSE;
  protections.T_podshipnika_reduktora_t1_HA.inOpcCommandsDisabled:=FALSE;
  protections.T_podshipnika_reduktora_t2_HA.inOpcCommandsDisabled:=FALSE;
  protections.T_podshipnika_reduktora_t3_HA.inOpcCommandsDisabled:=FALSE;
  protections.T_podshipnika_reduktora_t4_HA.inOpcCommandsDisabled:=FALSE;
  protections.T_opornogo_podshipnika_nagnetatelia_t1_HA.inOpcCommandsDisabled:=FALSE;
  protections.T_opornogo_podshipnika_nagnetatelia_t2_HA.inOpcCommandsDisabled:=FALSE;
  protections.T_opornogo_podshipnika_nagnetatelia_t3_HA.inOpcCommandsDisabled:=FALSE;
  protections.T_opornoupornogo_podshipnika_nagnetatelia_t4_HA.inOpcCommandsDisabled:=FALSE;
  protections.T_gaza_na_vykhode_nagnetatelia_HA.inOpcCommandsDisabled:=FALSE;
  protections.dP_maslogaz_LA.inOpcCommandsDisabled:=FALSE;
  protections.P_masla_smazki_nizkoe_LA.inOpcCommandsDisabled:=FALSE;
  protections.Vibratciia_STD_t1_HA.inOpcCommandsDisabled:=FALSE;
  protections.Vibratciia_STD_t2_HA.inOpcCommandsDisabled:=FALSE;
  protections.Vibratciia_rotora_nagnetatelia_t1_HA.inOpcCommandsDisabled:=FALSE;
  protections.Vibratciia_rotora_nagnetatelia_t2_HA.inOpcCommandsDisabled:=FALSE;
  protections.Vibratciia_rotora_nagnetatelia_t3_HA.inOpcCommandsDisabled:=FALSE;
  protections.Vibratciia_rotora_nagnetatelia_t4_HA.inOpcCommandsDisabled:=FALSE;
  protections.Osevoi_sdvig_rotora_nagnetatelia_HA.inOpcCommandsDisabled:=FALSE;
  protections.Uroven_masla_v_maslobake_LA.inOpcCommandsDisabled:=FALSE;
  protections.OsevojSdvigPravyjDi.inOpcCommandsDisabled:=FALSE;
  protections.OsevojSdvigLevyjDi.inOpcCommandsDisabled:=FALSE;
  protections.dP_masloGaz_LowDI.inOpcCommandsDisabled:=FALSE;
  protections.DavlenieMaslaSmazkiDi.inOpcCommandsDisabled:=FALSE;
  protections.mvOff.inOpcCommandsDisabled:=FALSE;
  protections.NeispravnostVozbuzhdenijaDi.inOpcCommandsDisabled:=FALSE;
  protections.AO_KC.inOpcCommandsDisabled:=FALSE;
  protections.AO_PRU.inOpcCommandsDisabled:=FALSE;
  protections.AO_SHU.inOpcCommandsDisabled:=FALSE;
  protections.Srab_BEAO.inOpcCommandsDisabled:=FALSE;
  protections.EAO_PRU.inOpcCommandsDisabled:=FALSE;
  protections.BEAO_knSHU.inOpcCommandsDisabled:=FALSE;
  protections.Kran1sdvig.inOpcCommandsDisabled:=FALSE;
  protections.Kran2sdvig.inOpcCommandsDisabled:=FALSE;
END_FUNCTION

FUNCTION_BLOCK fb_AlgoritmsManager
  VAR_IN_OUT
    str_AM : struct_AlgoritmsManager;
  END_VAR
  VAR
    onInit : BOOL;
  END_VAR
  VAR_EXTERNAL
    ai : AiConfig;
  END_VAR
  VAR
    EoTrig : R_TRIG;
    EoFTrig : F_TRIG;
    PsLampTrig : R_TRIG;
    PsLampFTrig : F_TRIG;
    Ring : R_TRIG;
    Line : R_TRIG;
    statusDualInput : TYPE_statusDualInput;
  END_VAR
  VAR_EXTERNAL
    IM : ImConfig;
    protections : ProtectionsConfig;
    algoritms : AlgoritmsConfig;
    ModeGpa : TYPE_ModeGpa;
  END_VAR

  IF NOT onInit THEN
            DisableAiLimits(ai);
            IM.SingleSignals.P_oil_low.Disabled_Sig:=TRUE;
            IM.SingleSignals.dP_oilgaz_low.Disabled_Sig:=TRUE;
            str_AM.nMode:=ModeGpa.MODE_STOP;
            BlockAllIM(IM);
            runIfNotRunning(algoritms.AutoTen);
  onInit:=TRUE;
  END_IF;

  str_AM.DiscretPS:=anyDiscretPS(IM);
  str_AM.AnalogsPs:=anyAnalogsPs(ai);
  str_AM.ProtectionSignaling:=anyProtectionSignaling(protections);

  EoTrig(CLK := IM.SingleSignals.BEO_Srabat.Q);
  IF EoTrig.Q THEN
  	stopPusk(algoritms);
  	resetAndDisable(algoritms.Remont);
  	resetAndDisable(algoritms.no);
  	resetAndDisable(algoritms.ao);
  	str_AM.nMode:=ModeGpa.MODE_EO;
  END_IF;
  EoFTrig(CLK := IM.SingleSignals.BEO_Srabat.Q);
  IF EoFTrig.Q THEN
  	str_AM.nMode:=ModeGpa.MODE_STOP;
  	runIfNotRunning(algoritms.ao);
  END_IF;

  IF (str_AM.ProtectionSignaling OR Im.SingleSignals.AO_KC.Q OR Im.SingleSignals.AOGPA_knopkaSHU.Q OR Im.SingleSignals.AOGPA_PRU.Q )
  	AND NOT((str_AM.mode=ModeGpa.MODE_AO) OR (str_AM.mode=ModeGpa.MODE_EO) OR IM.SingleOutputs.IndikicijaAS_fonar.Q
            OR (str_AM.mode=ModeGpa.MODE_TESTAZ) OR (str_AM.mode=ModeGpa.MODE_TESTDPMG) OR (str_AM.mode=ModeGpa.MODE_REMONT) OR
            (str_AM.mode=ModeGpa.MODE_TESTPMS))THEN
  		runIfNotRunning(algoritms.ao);
  	str_AM.nMode:=ModeGpa.MODE_AO;
  END_IF;

  IF Im.SingleSignals.NOGPA_knopkaSHU.Q  AND algoritms.no.CanRun THEN
  	runIfNotRunning(algoritms.no);
            str_AM.nMode:=ModeGpa.MODE_NO;
  END_IF;

  PsLampTrig(CLK := str_AM.DiscretPS OR str_AM.AnalogsPs);
  IF PsLampTrig.Q THEN
            runIfNotRunningSO(IM.SingleOutputs.IndikicijaPS_fonar);
  END_IF;
  PsLampFTrig(CLK := str_AM.DiscretPS OR str_AM.AnalogsPs);
  IF PsLampFTrig.Q THEN
            resetIfRunningSO(IM.SingleOutputs.IndikicijaPS_fonar);
  END_IF;

  IF str_AM.mode = ModeGpa.MODE_WORK_Line OR str_AM.mode = ModeGpa.MODE_WORK_Ring  THEN

  	Ring(CLK:=Im.kran6.onStatus=statusDualInput.STATUS_On);
  	Line(CLK:=Im.kran6.onStatus=statusDualInput.STATUS_Off);

  	IF Ring.Q AND str_AM.mode = ModeGpa.MODE_WORK_Line THEN
  		str_AM.nMode:=ModeGpa.MODE_WORK_Ring;
  	END_IF;
  	IF Line.Q AND str_AM.mode = ModeGpa.MODE_WORK_Ring THEN
  		str_AM.nMode:=ModeGpa.MODE_WORK_Line;
  	END_IF;

  END_IF;

  IF str_AM.mode = ModeGpa.MODE_WORK_Line THEN
            runIfNotRunning(alg:=algoritms.AntiPompag);
  	ELSE
            resetAndDisable(alg:=algoritms.AntiPompag);
  END_IF;

  IF str_AM.nMode<>str_AM.mode THEN
  	str_AM.mode:=str_AM.nMode;
  	CASE str_AM.mode OF
  	(*ModeGpa.MODE_REMONT*)1:
  		stopPusk(algoritms);
  		resetAndDisable(alg:=algoritms.no);
  		resetAndDisable(alg:=algoritms.ao);
  		resetAndDisable(alg:=algoritms.TestProtection);
                      resetAndDisable(alg:=algoritms.testIm);

  	(*ModeGpa.MODE_TESTAZ*)16:
  		stopPusk(algoritms);
  		resetAndDisable(alg:=algoritms.ao);
  		resetAndDisable(alg:=algoritms.no);
                      resetAndDisable(alg:=algoritms.Remont);
                      resetAndDisable(alg:=algoritms.testIm);

            (*ModeGpa.MODE_TESTIM*)15:
                      stopPusk(algoritms);
                      resetAndDisable(alg:=algoritms.Remont);
                      resetAndDisable(alg:=algoritms.TestProtection);

  	(*ModeGpa.MODE_EO*)14:
  		stopPusk(algoritms);
  		resetAndDisable(alg:=algoritms.no);
  		resetAndDisable(alg:=algoritms.ao);
  		resetAndDisable(alg:=algoritms.Remont);
                      resetAndDisable(alg:=algoritms.testIm);
                      resetAndDisable(alg:=algoritms.TestProtection);
  	(*ModeGpa.MODE_AO*)13:
  		(*//stopPusk();*)
  		resetAndDisable(alg:=algoritms.no);
  		resetAndDisable(alg:=algoritms.Remont);
                      resetAndDisable(alg:=algoritms.testIm);
                      resetAndDisable(alg:=algoritms.TestProtection);
                      algoritms.VibegPNS.inCanRun:=TRUE;
  	(*ModeGpa.MODE_NO*)12:
  		stopPusk(algoritms);
                      resetAndDisable(alg:=algoritms.testIm);
                      resetAndDisable(alg:=algoritms.Remont);
                      resetAndDisable(alg:=algoritms.TestProtection);
                      algoritms.VibegPNS.inCanRun:=TRUE;
  		algoritms.ao.inCanRun:=TRUE;
  	(*ModeGpa.MODE_APUSK*)8:
  		resetAndDisable(alg:=algoritms.SemiAutoPusk);
  		resetAndDisable(alg:=algoritms.puskV);
  		resetAndDisable(alg:=algoritms.puskK);
  		resetAndDisable(alg:=algoritms.testdPmg);
  		resetAndDisable(alg:=algoritms.testPms);
  		(*resetAndDisable(alg:=algoritms.testIm);
                      resetAndDisable(alg:=algoritms.TestProtection);
                      resetAndDisable(alg:=algoritms.Remont);*)
  		resetAndDisable(alg:=algoritms.ppu);
  		algoritms.no.inCanRun:=TRUE;
  		algoritms.ao.inCanRun:=TRUE;

  	(*ModeGpa.MODE_MPUSK*)9:
  		resetAndDisable(alg:=algoritms.Apusk);
  		resetAndDisable(alg:=algoritms.puskV);
  		resetAndDisable(alg:=algoritms.puskK);
  		resetAndDisable(alg:=algoritms.testdPmg);
  		resetAndDisable(alg:=algoritms.testPms);
  		(*resetAndDisable(alg:=algoritms.testIm);
                      resetAndDisable(alg:=algoritms.TestProtection);
                      resetAndDisable(alg:=algoritms.Remont);	*)
  		resetAndDisable(alg:=algoritms.ppu);
  		algoritms.no.inCanRun:=TRUE;
                      algoritms.no.inOpcCommandsDisabled:=FALSE;
  		algoritms.ao.inCanRun:=TRUE;
                      algoritms.ao.inOpcCommandsDisabled:=FALSE;

  	(*ModeGpa.MODE_PUSKK*)5:
                      resetAndDisable(alg:=algoritms.ppu);
  		resetAndDisable(alg:=algoritms.Apusk);
  		resetAndDisable(alg:=algoritms.SemiAutoPusk);
  		resetAndDisable(alg:=algoritms.TestProtection);
                      resetAndDisable(alg:=algoritms.Remont);
  		resetAndDisable(alg:=algoritms.testIm	 );
  		algoritms.no.inCanRun:=TRUE;
                      algoritms.no.inOpcCommandsDisabled:=FALSE;
  		algoritms.ao.inCanRun:=TRUE;
                      algoritms.ao.inOpcCommandsDisabled:=FALSE;
  	(*ModeGpa.MODE_PUSKV*)4:
                      resetAndDisable(alg:=algoritms.ppu);
  		resetAndDisable(alg:=algoritms.Apusk);
  		resetAndDisable(alg:=algoritms.SemiAutoPusk);
  		resetAndDisable(alg:=algoritms.TestProtection);
                      resetAndDisable(alg:=algoritms.Remont);
  		resetAndDisable(alg:=algoritms.testIm	 );
  		algoritms.no.inCanRun:=TRUE;
                      algoritms.no.inOpcCommandsDisabled:=FALSE;
  		algoritms.ao.inCanRun:=TRUE;
                      algoritms.ao.inOpcCommandsDisabled:=FALSE;

  	(*ModeGpa.MODE_TESTDPMG*)6:
                      resetAndDisable(alg:=algoritms.ppu);
  		resetAndDisable(alg:=algoritms.Apusk);
  		resetAndDisable(alg:=algoritms.SemiAutoPusk);
  		resetAndDisable(alg:=algoritms.TestProtection);
                      resetAndDisable(alg:=algoritms.Remont);
  		resetAndDisable(alg:=algoritms.testIm	 );
  		algoritms.no.inCanRun:=TRUE;
                      algoritms.no.inOpcCommandsDisabled:=FALSE;
  		algoritms.ao.inCanRun:=TRUE;
                      algoritms.ao.inOpcCommandsDisabled:=FALSE;

  	(*ModeGpa.MODE_TESTPMS*)7:
                      resetAndDisable(alg:=algoritms.ppu);
  		resetAndDisable(alg:=algoritms.Apusk);
  		resetAndDisable(alg:=algoritms.SemiAutoPusk);
  		resetAndDisable(alg:=algoritms.TestProtection);
                      resetAndDisable(alg:=algoritms.Remont);
  		resetAndDisable(alg:=algoritms.testIm);
  		algoritms.no.inCanRun:=TRUE;
                      algoritms.no.inOpcCommandsDisabled:=FALSE;
  		algoritms.ao.inCanRun:=TRUE;
                      algoritms.ao.inOpcCommandsDisabled:=FALSE;

  	(*ModeGpa.MODE_WORK_Ring*)10:
  		resetAndDisable(alg:=algoritms.Apusk);
  		resetAndDisable(alg:=algoritms.SemiAutoPusk);
  		resetAndDisable(alg:=algoritms.puskV);
  		resetAndDisable(alg:=algoritms.puskK);
  		resetAndDisable(alg:=algoritms.testdPmg);
  		resetAndDisable(alg:=algoritms.testPms);
  		resetAndDisable(alg:=algoritms.ppu);
  		algoritms.no.inCanRun:=TRUE;
                      algoritms.no.inOpcCommandsDisabled:=FALSE;
  		algoritms.ao.inCanRun:=TRUE;
                      algoritms.ao.inOpcCommandsDisabled:=FALSE;

  	(*ModeGpa.MODE_WORK_Line*)11:
  		resetAndDisable(alg:=algoritms.Apusk);
  		resetAndDisable(alg:=algoritms.SemiAutoPusk);
  		resetAndDisable(alg:=algoritms.puskV);
  		resetAndDisable(alg:=algoritms.puskK);
  		resetAndDisable(alg:=algoritms.testdPmg);
  		resetAndDisable(alg:=algoritms.testPms);
  		resetAndDisable(alg:=algoritms.ppu);
  		resetAndDisable(alg:=algoritms.testIm	 );
  		algoritms.no.inCanRun:=TRUE;
                      algoritms.no.inOpcCommandsDisabled:=FALSE;
  		algoritms.ao.inCanRun:=TRUE;
                      algoritms.ao.inOpcCommandsDisabled:=FALSE;

  	(*ModeGpa.MODE_STOP*)2:
  		algoritms.ppu.inCanRun:=TRUE;
                      runIfNotRunning(alg:=algoritms.ppu);
  		algoritms.no.inCanRun:=TRUE;
                      algoritms.no.inOpcCommandsDisabled:=FALSE;
  		algoritms.ao.inCanRun:=TRUE;
                      algoritms.ao.inOpcCommandsDisabled:=FALSE;
                      (*UnBlockAllProtections(protections);*)
  		BlockAllIM(IM);
  		algoritms.Remont.inCanRun:=TRUE;
  		algoritms.Remont.inOpcCommandsDisabled:=FALSE;
  		algoritms.testim.inCanRun:=TRUE;
  		algoritms.testim.inOpcCommandsDisabled:=FALSE;
  		algoritms.TestProtection.inCanRun:=TRUE;
  		algoritms.TestProtection.inOpcCommandsDisabled:=FALSE;
                      algoritms.VibegPNS.inCanRun:=FALSE;
                      algoritms.AutoAvom.inCanRun:=FALSE;
  		(*resetAndDisable(alg:=algoritms.puskV);
  		resetAndDisable(alg:=algoritms.puskK);
  		resetAndDisable(alg:=algoritms.testdPmg);
  		resetAndDisable(alg:=algoritms.testPms);*)
  	(*ModeGpa.MODE_READY*)3:
  		resetAndDisable(alg:=algoritms.Remont);
  		resetAndDisable(alg:=algoritms.testim);
  		resetAndDisable(alg:=algoritms.TestProtection);
                      algoritms.Apusk.inCanRun:=TRUE;
                      algoritms.Apusk.inOpcCommandsDisabled:=FALSE;
  		algoritms.SemiAutoPusk.inCanRun:=TRUE;
                      algoritms.SemiAutoPusk.inOpcCommandsDisabled:=FALSE;
  	END_CASE;
  END_IF;
END_FUNCTION_BLOCK

FUNCTION anyProtectionInRemont : BOOL
  VAR_INPUT
    protections : ProtectionsConfig;
  END_VAR

  anyProtectioninRemont:=
  protections.T_perednego_opornogo_podshipnika_dvigatelia_t1_HA.Remont OR
  protections.T_zadnego_opornogo_podshipnika_dvigatelia_t2_HA.Remont OR
  protections.T_podshipnika_reduktora_t1_HA.Remont OR
  protections.T_podshipnika_reduktora_t2_HA.Remont OR
  protections.T_podshipnika_reduktora_t3_HA.Remont OR
  protections.T_podshipnika_reduktora_t4_HA.Remont OR
  protections.T_opornogo_podshipnika_nagnetatelia_t1_HA.Remont OR
  protections.T_opornogo_podshipnika_nagnetatelia_t2_HA.Remont OR
  protections.T_opornogo_podshipnika_nagnetatelia_t3_HA.Remont OR
  protections.T_opornoupornogo_podshipnika_nagnetatelia_t4_HA.Remont OR
  protections.T_gaza_na_vykhode_nagnetatelia_HA.Remont OR
  protections.dP_maslogaz_LA.Remont OR
  protections.P_masla_smazki_nizkoe_LA.Remont OR
  protections.Vibratciia_STD_t1_HA.Remont OR
  protections.Vibratciia_STD_t2_HA.Remont OR
  protections.Vibratciia_rotora_nagnetatelia_t1_HA.Remont OR
  protections.Vibratciia_rotora_nagnetatelia_t2_HA.Remont OR
  protections.Vibratciia_rotora_nagnetatelia_t3_HA.Remont OR
  protections.Vibratciia_rotora_nagnetatelia_t4_HA.Remont OR
  protections.Osevoi_sdvig_rotora_nagnetatelia_HA.Remont OR
  protections.Uroven_masla_v_maslobake_LA.Remont OR
  protections.OsevojSdvigPravyjDi.Remont OR
  protections.OsevojSdvigLevyjDi.Remont OR
  protections.dP_masloGaz_LowDI.Remont OR
  protections.DavlenieMaslaSmazkiDi.Remont OR
  protections.mvOff.Remont OR
  protections.NeispravnostVozbuzhdenijaDi.Remont OR
  protections.AO_KC.Remont OR
  protections.AO_PRU.Remont OR
  protections.AO_SHU.Remont OR
  protections.Srab_BEAO.Remont OR
  protections.EAO_PRU.Remont OR
  protections.BEAO_knSHU.Remont OR
  protections.Kran1sdvig.Remont OR
  protections.Kran2sdvig.Remont;
END_FUNCTION

FUNCTION runAllProtections : BOOL
  VAR_IN_OUT
    protections : ProtectionsConfig;
  END_VAR

  runAiProtection(protections.T_perednego_opornogo_podshipnika_dvigatelia_t1_HA);
  runAiProtection(protections.T_zadnego_opornogo_podshipnika_dvigatelia_t2_HA);
  runAiProtection(protections.T_podshipnika_reduktora_t1_HA);
  runAiProtection(protections.T_podshipnika_reduktora_t2_HA);
  runAiProtection(protections.T_podshipnika_reduktora_t3_HA);
  runAiProtection(protections.T_podshipnika_reduktora_t4_HA);
  runAiProtection(protections.T_opornogo_podshipnika_nagnetatelia_t1_HA);
  runAiProtection(protections.T_opornogo_podshipnika_nagnetatelia_t2_HA);
  runAiProtection(protections.T_opornogo_podshipnika_nagnetatelia_t3_HA);
  runAiProtection(protections.T_opornoupornogo_podshipnika_nagnetatelia_t4_HA);
  runAiProtection(protections.T_gaza_na_vykhode_nagnetatelia_HA);
  runAiProtection(protections.dP_maslogaz_LA);
  runAiProtection(protections.P_masla_smazki_nizkoe_LA);
  runAiProtection(protections.Vibratciia_STD_t1_HA);
  runAiProtection(protections.Vibratciia_STD_t2_HA);
  runAiProtection(protections.Vibratciia_rotora_nagnetatelia_t1_HA);
  runAiProtection(protections.Vibratciia_rotora_nagnetatelia_t2_HA);
  runAiProtection(protections.Vibratciia_rotora_nagnetatelia_t3_HA);
  runAiProtection(protections.Vibratciia_rotora_nagnetatelia_t4_HA);
  runAiProtection(protections.Osevoi_sdvig_rotora_nagnetatelia_HA);
  runAiProtection(protections.Uroven_masla_v_maslobake_LA);

  runDiProtection(protections.OsevojSdvigPravyjDi);
  runDiProtection(protections.OsevojSdvigLevyjDi);
  runDiProtection(protections.dP_masloGaz_LowDI);
  runDiProtection(protections.DavlenieMaslaSmazkiDi);
  runDiProtection(protections.mvOff);
  runDiProtection(protections.NeispravnostVozbuzhdenijaDi);
  runDiProtection(protections.AO_KC);
  runDiProtection(protections.AO_PRU);
  runDiProtection(protections.AO_SHU);
  runDiProtection(protections.Srab_BEAO);
  runDiProtection(protections.EAO_PRU);
  runDiProtection(protections.BEAO_knSHU);
  runDiProtection(protections.Kran1sdvig);
  runDiProtection(protections.Kran2sdvig);
END_FUNCTION

FUNCTION ResetAllSignaling : BOOL
  VAR_IN_OUT
    protections : ProtectionsConfig;
  END_VAR

  IF protections.T_perednego_opornogo_podshipnika_dvigatelia_t1_HA.Signaling THEN
      resetAiProtection(protections.T_perednego_opornogo_podshipnika_dvigatelia_t1_HA);  END_IF;

  IF protections.T_zadnego_opornogo_podshipnika_dvigatelia_t2_HA.Signaling THEN
      resetAiProtection(protections.T_zadnego_opornogo_podshipnika_dvigatelia_t2_HA); END_IF;

  IF protections.T_podshipnika_reduktora_t1_HA.Signaling THEN
      resetAiProtection(protections.T_podshipnika_reduktora_t1_HA); END_IF;

  IF protections.T_podshipnika_reduktora_t2_HA.Signaling THEN
      resetAiProtection(protections.T_podshipnika_reduktora_t2_HA); END_IF;

  IF protections.T_podshipnika_reduktora_t3_HA.Signaling THEN
      resetAiProtection(protections.T_podshipnika_reduktora_t3_HA); END_IF;

  IF protections.T_podshipnika_reduktora_t4_HA.Signaling THEN
      resetAiProtection(protections.T_podshipnika_reduktora_t4_HA); END_IF;

  IF protections.T_opornogo_podshipnika_nagnetatelia_t1_HA.Signaling THEN
      resetAiProtection(protections.T_opornogo_podshipnika_nagnetatelia_t1_HA); END_IF;

  IF protections.T_opornogo_podshipnika_nagnetatelia_t2_HA.Signaling THEN
      resetAiProtection(protections.T_opornogo_podshipnika_nagnetatelia_t2_HA); END_IF;

  IF protections.T_opornogo_podshipnika_nagnetatelia_t3_HA.Signaling THEN
      resetAiProtection(protections.T_opornogo_podshipnika_nagnetatelia_t3_HA); END_IF;

  IF protections.T_opornoupornogo_podshipnika_nagnetatelia_t4_HA.Signaling THEN
      resetAiProtection(protections.T_opornoupornogo_podshipnika_nagnetatelia_t4_HA); END_IF;

  IF protections.T_gaza_na_vykhode_nagnetatelia_HA.Signaling THEN
      resetAiProtection(protections.T_gaza_na_vykhode_nagnetatelia_HA); END_IF;

  IF protections.dP_maslogaz_LA.Signaling THEN
     resetAiProtection(protections.dP_maslogaz_LA); END_IF;

  IF protections.P_masla_smazki_nizkoe_LA.Signaling THEN
      resetAiProtection(protections.P_masla_smazki_nizkoe_LA); END_IF;

  IF protections.Vibratciia_STD_t1_HA.Signaling THEN
      resetAiProtection(protections.Vibratciia_STD_t1_HA); END_IF;

  IF protections.Vibratciia_STD_t2_HA.Signaling THEN
      resetAiProtection(protections.Vibratciia_STD_t2_HA); END_IF;

  IF protections.Vibratciia_rotora_nagnetatelia_t1_HA.Signaling THEN
      resetAiProtection(protections.Vibratciia_rotora_nagnetatelia_t1_HA); END_IF;

  IF protections.Vibratciia_rotora_nagnetatelia_t2_HA.Signaling THEN
      resetAiProtection(protections.Vibratciia_rotora_nagnetatelia_t2_HA); END_IF;

  IF protections.Vibratciia_rotora_nagnetatelia_t3_HA.Signaling THEN
      resetAiProtection(protections.Vibratciia_rotora_nagnetatelia_t3_HA); END_IF;

  IF protections.Vibratciia_rotora_nagnetatelia_t4_HA.Signaling THEN
      resetAiProtection(protections.Vibratciia_rotora_nagnetatelia_t4_HA); END_IF;

  IF protections.Osevoi_sdvig_rotora_nagnetatelia_HA.Signaling THEN
      resetAiProtection(protections.Osevoi_sdvig_rotora_nagnetatelia_HA); END_IF;

  IF protections.Uroven_masla_v_maslobake_LA.Signaling THEN
      resetAiProtection(protections.Uroven_masla_v_maslobake_LA); END_IF;

  IF protections.OsevojSdvigPravyjDi.Signaling THEN
      resetDiProtection(protections.OsevojSdvigPravyjDi); END_IF;

  IF protections.OsevojSdvigLevyjDi.Signaling THEN
      resetDiProtection(protections.OsevojSdvigLevyjDi); END_IF;

  IF protections.dP_masloGaz_LowDI.Signaling THEN
      resetDiProtection(protections.dP_masloGaz_LowDI); END_IF;

  IF protections.DavlenieMaslaSmazkiDi.Signaling THEN
      resetDiProtection(protections.DavlenieMaslaSmazkiDi); END_IF;

  IF protections.mvOff.Signaling THEN
      resetDiProtection(protections.mvOff); END_IF;

  IF protections.NeispravnostVozbuzhdenijaDi.Signaling THEN
      resetDiProtection(protections.NeispravnostVozbuzhdenijaDi); END_IF;

  IF protections.AO_KC.Signaling THEN
      resetDiProtection(protections.AO_KC); END_IF;

  IF protections.AO_PRU.Signaling THEN
      resetDiProtection(protections.AO_PRU); END_IF;

  IF protections.AO_SHU.Signaling THEN
      resetDiProtection(protections.AO_SHU); END_IF;

  IF protections.Srab_BEAO.Signaling THEN
      resetDiProtection(protections.Srab_BEAO); END_IF;

  IF protections.EAO_PRU.Signaling THEN
      resetDiProtection(protections.EAO_PRU); END_IF;

  IF protections.BEAO_knSHU.Signaling THEN
      resetDiProtection(protections.BEAO_knSHU); END_IF;

  IF protections.Kran1sdvig.Signaling THEN
      resetDiProtection(protections.Kran1sdvig); END_IF;

  IF protections.Kran2sdvig.Signaling THEN
      resetDiProtection(protections.Kran2sdvig); END_IF;
END_FUNCTION

FUNCTION autoRunProtections : BOOL
  VAR_IN_OUT
    protections : ProtectionsConfig;
  END_VAR

  runAiProtection(protections.T_perednego_opornogo_podshipnika_dvigatelia_t1_HA);

      runAiProtection(protections.T_zadnego_opornogo_podshipnika_dvigatelia_t2_HA);

      runAiProtection(protections.T_podshipnika_reduktora_t1_HA);

      runAiProtection(protections.T_podshipnika_reduktora_t2_HA);

      runAiProtection(protections.T_podshipnika_reduktora_t3_HA);

      runAiProtection(protections.T_podshipnika_reduktora_t4_HA);

      runAiProtection(protections.T_opornogo_podshipnika_nagnetatelia_t1_HA);

      runAiProtection(protections.T_opornogo_podshipnika_nagnetatelia_t2_HA);

      runAiProtection(protections.T_opornogo_podshipnika_nagnetatelia_t3_HA);

      runAiProtection(protections.T_opornoupornogo_podshipnika_nagnetatelia_t4_HA);

      runAiProtection(protections.T_gaza_na_vykhode_nagnetatelia_HA);

      runAiProtection(protections.Osevoi_sdvig_rotora_nagnetatelia_HA);

      runAiProtection(protections.Uroven_masla_v_maslobake_LA);

      runDiProtection(protections.OsevojSdvigPravyjDi);

      runDiProtection(protections.OsevojSdvigLevyjDi);

      runDiProtection(protections.NeispravnostVozbuzhdenijaDi);

      runDiProtection(protections.AO_KC);

      runDiProtection(protections.AO_PRU);

      runDiProtection(protections.AO_SHU);

      runDiProtection(protections.Srab_BEAO);

      runDiProtection(protections.EAO_PRU);

      runDiProtection(protections.BEAO_knSHU);
END_FUNCTION

FUNCTION_BLOCK fb_ProtectionsManager
  VAR
    cmd : BYTE;
  END_VAR
  VAR_IN_OUT
    str_PM : struct_ProtectionsManager;
  END_VAR
  VAR
    lastCmd : BYTE;
    autoRunPriznak : BOOL;
    onInit : BOOL;
  END_VAR
  VAR_EXTERNAL
    protections : ProtectionsConfig;
  END_VAR
  VAR
    timerUnBlock : TON;
    timerAutoRun : TON;
    UnBlockPriznak : BOOL;
  END_VAR

  IF NOT onInit THEN

      autoRunProtections(protections);
  onInit:=TRUE;
  END_IF;

  str_PM.protectionInRemont:=anyProtectioninRemont(protections);

  cmd := str_PM.inCommand;

  IF cmd <> 0 AND lastCmd <> cmd then
                UnBlockPriznak:=TRUE;
  	CASE BYTE_TO_INT(cmd) OF

  		(*RestartAllSignaling*) 1: 	ResetAllSignaling(protections);
  				          autoRunPriznak:=TRUE;

  	        (*RestartAllProtections*) 2: 	ResetAllProtections(protections);
                                                    autoRunPriznak:=TRUE;

                        (*CheckProtections*)  3: 	RunAllProtections(protections);

  	         (*ResetAllProtections*)  4: 	ResetAllProtections(protections);

  	END_CASE;

  END_IF;
  lastCmd := cmd;
  timerUnBlock(IN:=UnBlockPriznak, PT:=T#1S);
  timerAutoRun(IN:=autoRunPriznak, PT:=T#500MS);

  IF timerAutoRun.Q THEN autoRunProtections(protections);
  END_IF;

  IF timerUnBlock.Q THEN
  lastCmd:= 0;
  str_PM.inCommand:=0;
  autoRunPriznak:=FALSE;
  UnBlockPriznak:=FALSE;
  END_IF;
END_FUNCTION_BLOCK

PROGRAM program0
  VAR
    SysTime : LREAL;
    preSysTime : LREAL;
    tmpCycle : LREAL;
    preSys_s : ULINT;
    preSys_ns : ULINT;
  END_VAR
  VAR
    systime_ns AT %IL0.10.11 : ULINT;
    systime_s AT %IL0.10.10 : ULINT;
  END_VAR
  VAR_EXTERNAL
    cur_Cycle : REAL;
    gStart_Tmr : REAL;
  END_VAR
  VAR
    Timings : fb_Timings;
    _init : BOOL := TRUE;
    life_count : UINT;
    AI_structs_ini : proc_AI_Init;
    AI_Proc : proc_AI;
    AO_structs_ini : proc_AO_Init;
    AO_Proc : proc_AO;
    DI_structs_ini : proc_DI_Init;
    DI_Proc : proc_DI;
    DO_structs_ini : proc_DO_Init;
    DO_Proc : proc_DO;
    ini_AI_OPC : OPC_AI_init;
    Get_AI_OPC : OPC_AI_get;
    Set_AI_OPC : OPC_AI_set;
    Get_protections_OPC : OPC_protections_get;
    Set_protections_OPC : OPC_protections_set;
    Get_algoritms_OPC : OPC_algoritms_set;
    Set_algoritms_OPC : OPC_algoritms_get;
    IM_structs_ini : proc_IM_Init;
    IM_Proc : proc_IM;
    Get_IM_OPC : OPC_IM_get;
    Set_IM_OPC : OPC_IM_set;
    Protections_structs_ini : proc_Protections_Init;
    Protections_Proc : proc_Protection;
    Algoritms_Proc : proc_algoritms;
    AlgoritmsManager : fb_AlgoritmsManager;
    ProtectionsManager : fb_ProtectionsManager;
  END_VAR
  VAR_EXTERNAL
    algManager : struct_AlgoritmsManager;
    protectManager : struct_ProtectionsManager;
  END_VAR

  (* Обработка времени. *)
  SysTime := ULINT_TO_LREAL(systime_s) + (1.0E-9 * ULINT_TO_LREAL(systime_ns));
  preSysTime := SysTime;
  tmpCycle := ULINT_TO_LREAL(systime_s - preSys_s) + 1.0E-9 * (ULINT_TO_LREAL(systime_ns) - ULINT_TO_LREAL(preSys_ns));
  cur_Cycle := LREAL_TO_REAL(tmpCycle);
  preSys_s := systime_s;
  preSys_ns := systime_ns;
  IF gStart_Tmr < 99999.9 THEN gStart_Tmr := gStart_Tmr + cur_Cycle; END_IF;
  Timings();

  IF  _init (*or external_init_ai *) then           (* Требуется инициализация структур и ФБ. *)
    (* Инициализация аналоговых входов. *)
      AI_structs_ini(init := TRUE);
      AI_Proc((*init := FALSE*));

    (* Инициализация дискретных входов. *)
      DI_structs_ini(init := TRUE);
      DI_Proc((*init := FALSE*));

      (* Инициализация аналоговых выходов. *)
  (*     AO_structs_ini(init := TRUE);
         AO_Proc(init := TRUE);*)

    (* Инициализация дискретных выходов. *)
      DO_structs_ini(init := TRUE);
      DO_Proc((*init := FALSE*));

     (* Инициализация ИМ. *)
      IM_structs_ini(init := TRUE);
      IM_Proc();

     (* Инициализация Защит *)
      Protections_structs_ini(init := TRUE);
      (*Protections_Proc();*)

       (* Стартовая инициализация OPC-тэгов элементами канальных структур. *)
          (*___________________AI______________________________________________________________________________*)
      ini_AI_OPC();

      _init := FALSE;

    ELSE                         (* Завершена инициализация структур и ФБ. *)

  (* Перенос OPC-тэгов в элементы структур каналов. *)
        (*___________________________________________AI________________________________________________*)
      Get_AI_OPC();
      Get_IM_OPC();
      Get_protections_OPC();
      Get_algoritms_OPC();

     (* Пересчёт защит САУ. *)
     ProtectionsManager(protectManager);

       (* Пересчёт алгоритмов САУ. *)
     AlgoritmsManager(algManager);

      (****               Опрос входов.              ****)
          (* Опрос аналоговых входов. *)
      AI_Proc((*init := FALSE*));

          (* Опрос дискретных входов. *)
      DI_Proc((*init := FALSE*));

      (****              Запись выходов.             ****)
          (* Запись аналоговых выходов. *)
  (*    AO_Proc(init := FALSE);*)

       (* Запись дискретных выходов. *)
      DO_Proc((*init := FALSE*));

      (****               Опрос ИМ              ****)
      IM_Proc();

      (****            Опрос Защит              ****)
      Protections_Proc();

      Algoritms_Proc();

  END_IF;

  (* Передача информации на верхний уровень по OPC UA протоколу. *)
    (* Передача состояний каналов AI. *)
  Set_AI_OPC();
  (* Передача состояний каналов ИМ. *)
  Set_IM_OPC();
  (* Передача состояний защит. *)
  Set_protections_OPC();
  (* Передача состояний алгоритмов. *)
  Set_algoritms_OPC();
END_PROGRAM

FUNCTION_BLOCK fb_DualStateIm
  VAR_INPUT
    statOn : BOOL;
    statOff : BOOL;
  END_VAR
  VAR_IN_OUT
    StrDs : struct_DualStateIm;
  END_VAR
  VAR_INPUT
    statOn_reliability : BOOL;
    statOff_reliability : BOOL;
    inNs : TYPE_ReliableBit;
    inAccident : TYPE_ReliableBit;
    inCommand : WORD;
  END_VAR
  VAR
    _statOn : BOOL;
    _statOff : BOOL;
    getSdvig : BOOL;
    lastOnStatus : BYTE;
    cmd : BYTE;
    source : BYTE;
    lastCmd : BYTE;
    source_for_Status : BYTE;
    cmd_for_Status : BYTE;
    command_error_for_Status : BYTE;
    _sunpackerCommand : fb_sunpackerCommand;
    _statusDualInput : TYPE_statusDualInput;
    _commandDualInput : TYPE_commandDualInput;
    _commandErrorTimer : BOOL;
    onInit : BOOL := FALSE;
    resetErrorTimer : BOOL;
    _changWithoutCommand : BOOL;
    errorCMDTimer : TON;
    sdvigReset : TON;
    _errorReset : TON;
  END_VAR
  VAR_IN_OUT
    cmdOn : BOOL;
  END_VAR
  VAR_OUTPUT
    cmdOff : BOOL;
  END_VAR

  IF NOT onInit THEN
  IF StrDs.ISVALIDREF_cmdOn XOR StrDs.ISVALIDREF_cmdOff THEN
  	IF 	StrDs.ISVALIDREF_cmdOn THEN
  		lastCmd:= 2; (*baseCmdOff*)
  	ELSE
  		lastCmd:= 1; (*baseCmdOn*)
  	END_IF;
  END_IF;
  onInit:=TRUE;
  END_IF;

  (* ---- Если управление с ВУ заблокировано, то в ИМ передаем команду из алгоритма ---- *)
  IF StrDs.inOpcCommandsDisabled THEN
  	StrDs.inCommand := StrDs.inCommand_Alg;
  ELSE (* иначе передаем команду с АРМа*)
  	StrDs.inCommand := StrDs.inCommand_ARM;
  END_IF;

  (* ---- Формирование состояния механизма ---- *)

  IF (StrDs.ISVALIDREF_statOn) OR (StrDs.ISVALIDREF_statOff) THEN
  	IF (StrDs.ISVALIDREF_statOn) AND (StrDs.ISVALIDREF_statOff) THEN
  	StrDs.reliability:= statOn_reliability AND statOff_reliability;
  		_statOn  := statOn;
  		_statOff := statOff;
  	ELSIF (StrDs.ISVALIDREF_statOn) THEN
                       StrDs.reliability:= statOn_reliability;
  		_statOn  := statOn;
  		_statOff := NOT statOn;
  	ELSIF (StrDs.ISVALIDREF_statOff) THEN
  		 StrDs.reliability:= statOff_reliability;
  		_statOn  := NOT statOff;
  		_statOff :=statOff;
  	END_IF;

  	IF StrDs.reliability THEN
  		IF _statOn AND NOT _statOff 		THEN 	StrDs.onStatus := _statusDualInput.STATUS_ON;
  		ELSIF _statOff AND NOT _statOn 	THEN 	StrDs.onStatus := _statusDualInput.Status_OFF;
  		ELSIF NOT _statOn AND NOT _statOff 	THEN 	StrDs.onStatus := _statusDualInput.STATUS_TRANSITIONAL;
  		ELSE					StrDs.onStatus := _statusDualInput.STATUS_ERROR;
                      END_IF;

  	ELSE
  		StrDs.onStatus := _statusDualInput.STATUS_NOTDEFINED;

  	END_IF;
  ELSE
  	CASE BYTE_TO_INT(lastCmd) OF
  		(*baseCmdOn*) 1: StrDs.onStatus  := _statusDualInput.STATUS_ON;
  		(*baseCmdOff*) 2: StrDs.onStatus  := _statusDualInput.STATUS_OFF;

  	ELSE
  		 StrDs.onStatus := _statusDualInput.STATUS_NOTDEFINED;

  	END_CASE;
  END_IF;

  (* ---- Формирование признака сдвига ---- *)
  getSdvig := FALSE;
  IF (StrDs.ISVALIDREF_cmdOn OR StrDs.ISVALIDREF_cmdOff) THEN
  	IF NOT (StrDs.CmdOn OR StrDs.CmdOff) THEN
                       IF (lastOnStatus <> StrDs.onStatus AND
  		(StrDs.onStatus <> _statusDualInput.STATUS_NOTDEFINED AND
                       StrDs.onStatus <> _statusDualInput.STATUS_ERROR)     AND
  		(lastOnStatus <> _statusDualInput.STATUS_NOTDEFINED   AND
                       lastOnStatus <> _statusDualInput.STATUS_ERROR))
                      THEN
  			getSdvig   := TRUE;
  		END_IF;
  	END_IF;
  END_IF;

  IF getSdvig THEN StrDs.sdvig:= TRUE; END_IF;

  sdvigReset(IN:=StrDs.sdvig, PT:=T#15S);

  IF sdvigReset.Q THEN StrDs.sdvig:=FALSE; END_IF;

  lastOnStatus := StrDs.onStatus;

  StrDs.Accident := inAccident.value AND inAccident.reliability;
  StrDs.Ns := inNs.value AND inNs.reliability;
  StrDs.OpcCommandsDisabled := StrDs.inOpcCommandsDisabled;

  (* ---- Распаковка команды ---- *)
  _sunpackerCommand(command := StrDs.inCommand);
  	cmd := _sunpackerCommand.cmd;
  	source := _sunpackerCommand.source;

  (* ---- Обработка команды ---- *)
  IF cmd <> 0 AND lastCmd <> cmd and (((NOT StrDs.opcCommandsDisabled) AND source > 0) OR source = 0) then
  	CASE BYTE_TO_INT(cmd) OF
  	(*cmd_open*) 1 :
  			IF  StrDs.ISVALIDREF_cmdOn THEN StrDs.CmdOn := TRUE;
  				IF StrDs.ISVALIDREF_cmdOff THEN StrDs.CmdOff := FALSE; END_IF;
  			ELSIF  StrDs.ISVALIDREF_cmdOff THEN StrDs.CmdOff := FALSE;  END_IF;
  			errorCMDTimer(IN := false);
  			_commandErrorTimer := true;
  			StrDs.lastCmdIsOn := true;
  	(*cmd_close*) 2 :
  			IF StrDs.ISVALIDREF_cmdOff THEN StrDs.CmdOff := TRUE;
  				IF StrDs.ISVALIDREF_cmdOn THEN StrDs.CmdOn := FALSE; END_IF;
  			ELSIF StrDs.ISVALIDREF_cmdOn THEN StrDs.CmdOn := FALSE; END_IF;
  			errorCMDTimer(IN := false);
  			_commandErrorTimer := true;
  			StrDs.lastCmdIsOn := false;
  	(*cmd_reset*) 3 :    IF StrDs.ISVALIDREF_statOn OR StrDs.ISVALIDREF_statOff THEN
  			StrDs.CmdOn := FALSE;
  			StrDs.CmdOff := FALSE;
                                lastCmd :=0;
  			_commandErrorTimer := false;
  			StrDs.lastCmdIsOn := false;
                                END_IF;
  	END_CASE;
  	source_for_Status := source;
  	cmd_for_Status := cmd;
  	command_error_for_Status := 0;
  END_IF;

  lastCmd := cmd;
  errorCMDTimer(In := _commandErrorTimer, PT :=T#10s);

  (* ---- алгоритм  для команды ВКЛючить ---- *)
  IF (StrDs.onStatus = _statusDualInput.STATUS_ON) and (lastCmd = _commandDualInput.CMD_ON) then
  	IF StrDs.ISVALIDREF_cmdOn AND StrDs.ISVALIDREF_cmdOff then  StrDs.cmdOn := false; END_IF;

  	 errorCMDTimer(In := false);
  	 _commandErrorTimer := false;
  	 cmd_for_Status := 0;
  	 source_for_Status := 0;
  END_IF;

  (* ---- off ---- *)
  IF (StrDs.onStatus = _statusDualInput.STATUS_OFF) and (lastCmd = _commandDualInput.CMD_OFF) then
  	IF StrDs.ISVALIDREF_cmdOn AND StrDs.ISVALIDREF_cmdOff then  StrDs.cmdOff := false; END_IF;

  	 errorCMDTimer(In := false);
  	 _commandErrorTimer := false;
  	 cmd_for_Status := 0;
  	 source_for_Status := 0;
  END_IF;

  (* ---- ошибка исполнения команды ---- *)
  if errorCMDTimer.Q and (cmd_for_Status <> 0) then
  	command_error_for_Status :=  cmd_for_Status;
  	_commandErrorTimer := false;
  	StrDs.CmdOn := false;
  	StrDs.CmdOff := false;
  	lastCmd := 0;
  end_if;

  (* ---- сброс ошибки команды ---- *)
  StrDs.CommandFault := command_error_for_Status <> 0;
  _errorReset(IN := command_error_for_Status <> 0, PT := T#15S);
  IF _errorReset.Q THEN
  	cmd_for_Status := 0;
  	source_for_Status := 0;
  	command_error_for_Status := 0;
  END_IF;

  cmdOn := StrDs.cmdOn;
  cmdOff:= StrDs.cmdOff;

  (* ---- формирование зашифрованного статуса для АРМа ---- *)
  StrDs.status := shl(BYTE_TO_DWORD(source_for_Status), 29)
  		OR shl(BYTE_TO_DWORD(cmd_for_Status), 26)
  		OR shl(BYTE_TO_DWORD(command_error_for_Status), 23)
  		OR shl(bool_to_DWORD(StrDs.sdvig), 22)
  		OR shl(bool_to_DWORD(StrDs.OpcCommandsDisabled), 21)
  		OR shl(BOOL_TO_DWORD(StrDs.Ns), 4)
                  	OR shl(BOOL_TO_DWORD(StrDs.Accident ),3)
  		OR BYTE_TO_DWORD(StrDs.onStatus);
END_FUNCTION_BLOCK

FUNCTION_BLOCK fb_BaseProtection
  VAR_INPUT
    inSignaling : BOOL;
    inTag : BYTE;
    inRunOnStart : BOOL;
    inCanRun : BOOL;
    inHasError : BOOL;
    inEnded : BOOL;
    inOpcCommandsDisabled : BOOL;
    inCommand : WORD;
  END_VAR
  VAR_OUTPUT
    Tag : BYTE;
    status : DWORD;
    CanRun : BOOL;
    OpcCommandsDisabled : BOOL;
    isRunning : BOOL;
    HasError : BOOL;
    isEnded : BOOL;
    Remont : BOOL;
    Check : BOOL;
    Signaling : BOOL;
    SignalingTP : BOOL;
    RunOnStart : BOOL;
  END_VAR
  VAR
    _sunpackerCommand : fb_sunpackerCommand;
    _ProtectionTags : TYPE_ProtectionTags;
    _signalingTp : TOF;
    source : BYTE;
    cmd : BYTE;
    lastCmd : BYTE;
    source_for_Status : BYTE;
    cmd_for_Status : BYTE;
    command_error_for_Status : BYTE;
    resetCmdTimer : TON;
    resetCmdTimerPriznak : BOOL;
    signalinTimer : TON;
    runOnStart_Trig : R_TRIG;
  END_VAR

  Tag := inTag;
  RunOnStart := inRunOnStart;

  CanRun := inCanRun;
  hasError := inHasError;
  isEnded := inEnded;

  OpcCommandsDisabled := inOpcCommandsDisabled;

  _sunpackerCommand(command := inCommand);
  	source := _sunpackerCommand.source;
  	cmd := _sunpackerCommand.cmd;

  IF cmd <> 0 AND lastCmd <> cmd AND (((NOT opcCommandsDisabled) AND source > 0) OR source = 0) then
  	CASE BYTE_TO_INT(cmd) OF
  		(*cmdRun*) 1: 	IF CanRun AND NOT Remont THEN
  					isEnded := FALSE;
  					hasError 	:= FALSE;
  					isRunning := TRUE;
  					cmd_for_Status := cmd;
  					source_for_Status := source;
  					command_error_for_Status := 0;
  				ELSE
  					isRunning := FALSE;
  					isEnded := FALSE;
  					hasError 	:= FALSE;

  					cmd_for_Status := 0;
  					source_for_Status := source;
  					command_error_for_Status := cmd;
  				END_IF;
  		(*cmdReset*) 2: 	isRunning := FALSE;
  				isEnded := FALSE;
  				hasError 	:= FALSE;
  				inSignaling := FALSE;
  				Check := FALSE;
  				cmd_for_Status := cmd;
  				source_for_Status := source;
  				command_error_for_Status := 0;
  	(*cmd_setRemont*) 4 :	Remont := TRUE;
  				isRunning := FALSE;

  				cmd_for_Status := cmd;
  				source_for_Status := source;
  				command_error_for_Status := 0;
  	(*cmd_resetRemont*) 5 : 	IF inSignaling THEN
  					cmd_for_Status := 0;
  					source_for_Status := 0;
  					command_error_for_Status := cmd;
  				ELSE
  					Remont := FALSE;
  					isRunning := TRUE;

  					cmd_for_Status := cmd;
  					source_for_Status := source;
  					command_error_for_Status := 0;
  				END_IF;
  	(*cmd_setCheck*) 6 : 	Check := TRUE;

  				cmd_for_Status := cmd;
  				source_for_Status := source;
  				command_error_for_Status := 0;
  	END_CASE;
  	resetCmdTimer(IN := false);
  	resetCmdTimerPriznak := TRUE;
  END_IF;
  lastCmd := cmd;

  resetCmdTimer(IN := resetCmdTimerPriznak);
  IF resetCmdTimer.Q THEN
  	resetCmdTimerPriznak := FALSE;
  	source_for_Status := 0;
  	cmd_for_Status := 0;
  	command_error_for_Status := 0;
  END_IF;

  IF isRunning THEN
  	Signaling := inSignaling;
  	SignalingTP := _signalingTp.Q;
  ELSE
  	Signaling := 0;
  	SignalingTP := 0;
  END_IF;

  IF NOT Remont AND NOT Check THEN
  	_signalingTp(in := Signaling, PT := T#1s);
  ELSE
  	_signalingTp(in := FALSE);
  END_IF;

  status :=  SHL(BYTE_TO_DWORD(source_for_Status), 29)
  			OR SHL(BYTE_TO_DWORD(cmd_for_Status), 26)
  			OR SHL(BYTE_TO_DWORD(command_error_for_Status), 23)
  			OR SHL(BOOL_TO_DWORD(OpcCommandsDisabled ), 21)
  			OR SHL(BOOL_TO_DWORD(Signaling), 16)
  			OR SHL(BOOL_TO_DWORD(RunOnStart ), 15)
  			OR SHL(BOOL_TO_DWORD(remont), 6)
  			OR SHL(BOOL_TO_DWORD(Check), 5)
  			OR SHL(BOOL_TO_DWORD(hasError), 4)
  			OR SHL(BOOL_TO_DWORD(SignalingTP), 3)
  			OR SHL(BOOL_TO_DWORD(CanRun), 2)
  			OR SHL(BOOL_TO_DWORD(isEnded), 1)
  			OR BOOL_TO_DWORD(isRunning);
END_FUNCTION_BLOCK

FUNCTION_BLOCK fb_BaseAlgoritm
  VAR_IN_OUT
    StrAlg : struct_Alg;
  END_VAR
  VAR
    _sunpackerCommand : fb_sunpackerCommand;
    source : BYTE;
    cmd : BYTE;
    lastCmd : BYTE;
    source_for_Status : BYTE;
    cmd_for_Status : BYTE;
    command_error_for_Status : BYTE;
    resetCmdTimer : TON;
    resetCmdTimerPriznak : BOOL;
  END_VAR

  StrAlg.CanRun := StrAlg.inCanRun;
  StrAlg.hasError := StrAlg.inHasError OR (command_error_for_Status <> 0);
  StrAlg.isEnded := StrAlg.inEnded;

  StrAlg.OpcCommandsDisabled := StrAlg.inOpcCommandsDisabled;

  (* ---- Если управление с ВУ заблокировано, то передаем команду из алгоритма ---- *)
  IF StrAlg.inOpcCommandsDisabled THEN
  	StrAlg.inCommand := StrAlg.inCommand_Alg;
  ELSE (* иначе передаем команду с АРМа*)
  	StrAlg.inCommand := StrAlg.inCommand_ARM;
  END_IF;

  _sunpackerCommand(command := StrAlg.inCommand);
  	source := _sunpackerCommand.source;
  	cmd := _sunpackerCommand.cmd;

  IF cmd <> 0 AND lastCmd <> cmd AND (((NOT StrAlg.opcCommandsDisabled) AND source > 0) OR source = 0) then
  	CASE BYTE_TO_INT(cmd) OF
  		(*cmdRun*) 1: 	IF (StrAlg.CanRun) THEN
  					StrAlg.isRuning := TRUE;
  					StrAlg.isEnded := FALSE;
  					StrAlg.hasError 	:= FALSE;

  					cmd_for_Status := cmd;
  					source_for_Status := source;
  					command_error_for_Status := 0;
  				ELSE
  					StrAlg.isRuning := FALSE;
  					StrAlg.isEnded := FALSE;
  					StrAlg.hasError 	:= FALSE;

  					cmd_for_Status := 0;
  					source_for_Status := source;
  					command_error_for_Status := cmd;
  				END_IF;
  		(*cmdReset*) 2: 	StrAlg.isRuning := FALSE;
  				StrAlg.isEnded := FALSE;
  				StrAlg.hasError 	:= FALSE;
  				cmd_for_Status := cmd;
  				source_for_Status := source;
  				command_error_for_Status := 0;
  	END_CASE;
  	resetCmdTimer(IN := false);
  	resetCmdTimerPriznak := TRUE;
  END_IF;
  lastCmd := cmd;

  resetCmdTimer(IN := resetCmdTimerPriznak, PT := T#5S);
  IF resetCmdTimer.Q THEN
  	resetCmdTimerPriznak := FALSE;
  	source_for_Status := 0;
  	cmd_for_Status := 0;
  	command_error_for_Status := 0;
  END_IF;

  StrAlg.status :=  SHL(BYTE_TO_DWORD(source_for_Status), 29)
  			OR SHL(BYTE_TO_DWORD(cmd_for_Status), 26)
  			OR SHL(BYTE_TO_DWORD(command_error_for_Status), 23)
  			OR SHL(BOOL_TO_DWORD(StrAlg.OpcCommandsDisabled ), 21)
  			OR SHL(BOOL_TO_DWORD(StrAlg.hasError),4)
  			OR SHL(BOOL_TO_DWORD(StrAlg.CanRun),2)
  			OR SHL(BOOL_TO_DWORD(StrAlg.isEnded),1)
  			OR BOOL_TO_DWORD(StrAlg.isRuning);
END_FUNCTION_BLOCK

FUNCTION remontAllProtections : BOOL
  VAR_IN_OUT
    protections : ProtectionsConfig;
  END_VAR
  VAR CONSTANT
    cmdRemont : WORD := 4;
  END_VAR

  protections.T_perednego_opornogo_podshipnika_dvigatelia_t1_HA.inCommand_Alg:=cmdRemont;
  protections.T_zadnego_opornogo_podshipnika_dvigatelia_t2_HA.inCommand_Alg:=cmdRemont;
  protections.T_podshipnika_reduktora_t1_HA.inCommand_Alg:=cmdRemont;
  protections.T_podshipnika_reduktora_t2_HA.inCommand_Alg:=cmdRemont;
  protections.T_podshipnika_reduktora_t3_HA.inCommand_Alg:=cmdRemont;
  protections.T_podshipnika_reduktora_t4_HA.inCommand_Alg:=cmdRemont;
  protections.T_opornogo_podshipnika_nagnetatelia_t1_HA.inCommand_Alg:=cmdRemont;
  protections.T_opornogo_podshipnika_nagnetatelia_t2_HA.inCommand_Alg:=cmdRemont;
  protections.T_opornogo_podshipnika_nagnetatelia_t3_HA.inCommand_Alg:=cmdRemont;
  protections.T_opornoupornogo_podshipnika_nagnetatelia_t4_HA.inCommand_Alg:=cmdRemont;
  protections.T_gaza_na_vykhode_nagnetatelia_HA.inCommand_Alg:=cmdRemont;
  protections.dP_maslogaz_LA.inCommand_Alg:=cmdRemont;
  protections.P_masla_smazki_nizkoe_LA.inCommand_Alg:=cmdRemont;
  protections.Vibratciia_STD_t1_HA.inCommand_Alg:=cmdRemont;
  protections.Vibratciia_STD_t2_HA.inCommand_Alg:=cmdRemont;
  protections.Vibratciia_rotora_nagnetatelia_t1_HA.inCommand_Alg:=cmdRemont;
  protections.Vibratciia_rotora_nagnetatelia_t2_HA.inCommand_Alg:=cmdRemont;
  protections.Vibratciia_rotora_nagnetatelia_t3_HA.inCommand_Alg:=cmdRemont;
  protections.Vibratciia_rotora_nagnetatelia_t4_HA.inCommand_Alg:=cmdRemont;
  protections.Osevoi_sdvig_rotora_nagnetatelia_HA.inCommand_Alg:=cmdRemont;
  protections.Uroven_masla_v_maslobake_LA.inCommand_Alg:=cmdRemont;
  protections.OsevojSdvigPravyjDi.inCommand_Alg:=cmdRemont;
  protections.OsevojSdvigLevyjDi.inCommand_Alg:=cmdRemont;
  protections.dP_masloGaz_LowDI.inCommand_Alg:=cmdRemont;
  protections.DavlenieMaslaSmazkiDi.inCommand_Alg:=cmdRemont;
  protections.mvOff.inCommand_Alg:=cmdRemont;
  protections.NeispravnostVozbuzhdenijaDi.inCommand_Alg:=cmdRemont;
  protections.AO_KC.inCommand_Alg:=cmdRemont;
  protections.AO_PRU.inCommand_Alg:=cmdRemont;
  protections.AO_SHU.inCommand_Alg:=cmdRemont;
  protections.Srab_BEAO.inCommand_Alg:=cmdRemont;
  protections.EAO_PRU.inCommand_Alg:=cmdRemont;
  protections.BEAO_knSHU.inCommand_Alg:=cmdRemont;
  protections.Kran1sdvig.inCommand_Alg:=cmdRemont;
  protections.Kran2sdvig.inCommand_Alg:=cmdRemont;
END_FUNCTION

FUNCTION BlockAllProtections : BOOL
  VAR_IN_OUT
    protections : ProtectionsConfig;
  END_VAR

  protections.T_perednego_opornogo_podshipnika_dvigatelia_t1_HA.inOpcCommandsDisabled:=TRUE;
  protections.T_zadnego_opornogo_podshipnika_dvigatelia_t2_HA.inOpcCommandsDisabled:=TRUE;
  protections.T_podshipnika_reduktora_t1_HA.inOpcCommandsDisabled:=TRUE;
  protections.T_podshipnika_reduktora_t2_HA.inOpcCommandsDisabled:=TRUE;
  protections.T_podshipnika_reduktora_t3_HA.inOpcCommandsDisabled:=TRUE;
  protections.T_podshipnika_reduktora_t4_HA.inOpcCommandsDisabled:=TRUE;
  protections.T_opornogo_podshipnika_nagnetatelia_t1_HA.inOpcCommandsDisabled:=TRUE;
  protections.T_opornogo_podshipnika_nagnetatelia_t2_HA.inOpcCommandsDisabled:=TRUE;
  protections.T_opornogo_podshipnika_nagnetatelia_t3_HA.inOpcCommandsDisabled:=TRUE;
  protections.T_opornoupornogo_podshipnika_nagnetatelia_t4_HA.inOpcCommandsDisabled:=TRUE;
  protections.T_gaza_na_vykhode_nagnetatelia_HA.inOpcCommandsDisabled:=TRUE;
  protections.dP_maslogaz_LA.inOpcCommandsDisabled:=TRUE;
  protections.P_masla_smazki_nizkoe_LA.inOpcCommandsDisabled:=TRUE;
  protections.Vibratciia_STD_t1_HA.inOpcCommandsDisabled:=TRUE;
  protections.Vibratciia_STD_t2_HA.inOpcCommandsDisabled:=TRUE;
  protections.Vibratciia_rotora_nagnetatelia_t1_HA.inOpcCommandsDisabled:=TRUE;
  protections.Vibratciia_rotora_nagnetatelia_t2_HA.inOpcCommandsDisabled:=TRUE;
  protections.Vibratciia_rotora_nagnetatelia_t3_HA.inOpcCommandsDisabled:=TRUE;
  protections.Vibratciia_rotora_nagnetatelia_t4_HA.inOpcCommandsDisabled:=TRUE;
  protections.Osevoi_sdvig_rotora_nagnetatelia_HA.inOpcCommandsDisabled:=TRUE;
  protections.Uroven_masla_v_maslobake_LA.inOpcCommandsDisabled:=TRUE;
  protections.OsevojSdvigPravyjDi.inOpcCommandsDisabled:=TRUE;
  protections.OsevojSdvigLevyjDi.inOpcCommandsDisabled:=TRUE;
  protections.dP_masloGaz_LowDI.inOpcCommandsDisabled:=TRUE;
  protections.DavlenieMaslaSmazkiDi.inOpcCommandsDisabled:=TRUE;
  protections.mvOff.inOpcCommandsDisabled:=TRUE;
  protections.NeispravnostVozbuzhdenijaDi.inOpcCommandsDisabled:=TRUE;
  protections.AO_KC.inOpcCommandsDisabled:=TRUE;
  protections.AO_PRU.inOpcCommandsDisabled:=TRUE;
  protections.AO_SHU.inOpcCommandsDisabled:=TRUE;
  protections.Srab_BEAO.inOpcCommandsDisabled:=TRUE;
  protections.EAO_PRU.inOpcCommandsDisabled:=TRUE;
  protections.BEAO_knSHU.inOpcCommandsDisabled:=TRUE;
  protections.Kran1sdvig.inOpcCommandsDisabled:=TRUE;
  protections.Kran2sdvig.inOpcCommandsDisabled:=TRUE;
END_FUNCTION

FUNCTION_BLOCK ph_SingleOutput
  VAR_IN_OUT
    im : struct_singleOutput;
  END_VAR
  VAR_INPUT
    WhatCanIdo : BOOL;
    PhaseNumber : UINT;
  END_VAR
  VAR_IN_OUT
    StrPh : struct_PhaseAlgoritm;
  END_VAR
  VAR
    reset_Trig : R_TRIG;
  END_VAR

  IF StrPh.run AND NOT StrPh.start THEN
  	StrPh.start := TRUE;
  	StrPh.top := FALSE;
  	StrPh.error := FALSE;
            StrPh.run:=FALSE;

  	IF (WhatCanIdo) THEN
  	runIfNotRunningSO(im);
            ELSE
  	resetIfRunningSO(im);
            END_IF;
  END_IF;

  IF StrPh.start AND NOT StrPh.top THEN
  StrPh.top := (im.Q = WhatCanIdo);
  END_IF;

  reset_Trig(CLK := StrPh.reset);
  IF reset_Trig.Q THEN
  	StrPh.start := FALSE;
  	StrPh.error := FALSE;
  	StrPh.top := FALSE;
            StrPh.run:=FALSE;
            StrPh.reset:=FALSE;
  END_IF;

  StrPh.startStatus := SHL(BOOL_TO_DWORD(StrPh.start), PhaseNumber);
  StrPh.errorStatus := SHL(BOOL_TO_DWORD(StrPh.error), PhaseNumber);
  StrPh.topStatus := SHL(BOOL_TO_DWORD(StrPh.top), PhaseNumber);
END_FUNCTION_BLOCK

FUNCTION_BLOCK ph_SingleSignal
  VAR_IN_OUT
    im : struct_singleSignal;
  END_VAR
  VAR_INPUT
    expectedValue : BOOL := TRUE;
    PhaseNumber : UINT;
  END_VAR
  VAR_IN_OUT
    StrPh : struct_PhaseAlgoritm;
  END_VAR
  VAR
    reset_Trig : R_TRIG;
  END_VAR

  IF StrPh.run AND NOT StrPh.start THEN
  	StrPh.start := TRUE;
  	StrPh.top := FALSE;
  	StrPh.error := FALSE;
            StrPh.run:=FALSE;
  END_IF;

  IF StrPh.start AND NOT StrPh.top THEN
  StrPh.error:= NOT Im.reliability;
  StrPh.top := (Im.Q = expectedValue) AND (Im.reliability);
  END_IF;

  reset_Trig(CLK := StrPh.reset);
  IF reset_Trig.Q THEN
  	StrPh.start := FALSE;
  	StrPh.error := FALSE;
  	StrPh.top := FALSE;
            StrPh.run:=FALSE;
            StrPh.reset:=FALSE;
  END_IF;

  StrPh.startStatus := SHL(BOOL_TO_DWORD(StrPh.start), PhaseNumber);
  StrPh.errorStatus := SHL(BOOL_TO_DWORD(StrPh.error), PhaseNumber);
  StrPh.topStatus := SHL(BOOL_TO_DWORD(StrPh.top), PhaseNumber);
END_FUNCTION_BLOCK

FUNCTION_BLOCK ExtNarabotka
  VAR
    saveInterval : TIME := T#30S;
    narabotka : UDINT;
    timer : RTC;
    saveTimer : TON;
  END_VAR
  VAR_IN_OUT
    retain_narabotka : UDINT;
  END_VAR
  VAR
    initialized : BOOL;
  END_VAR
  VAR_INPUT
    started : BOOL;
    reset : BOOL;
  END_VAR

  IF NOT initialized THEN
  	narabotka:=retain_narabotka;
  	initialized:=TRUE;
  END_IF;

  timer();

  IF timer.Q THEN
  	narabotka:=DT_TO_UDINT( timer.CDT);

  END_IF;
  saveTimer(IN:=TRUE, PT:=saveInterval);
  IF saveTimer.Q THEN
  	retain_narabotka:=narabotka;
  	saveTimer(IN:=FALSE);
  END_IF;

  IF started THEN
  	IF NOT timer.Q THEN
  		timer.PDT:=UDINT_TO_DT(narabotka);
                      timer.IN:=TRUE;
  	END_IF;
  ELSE
  	IF timer.Q THEN
  		timer.IN:=FALSE;
                      saveTimer.IN:=FALSE;
  	END_IF;
  END_IF;

  IF reset THEN
  timer.PDT:=UINT_TO_DT(0);
  IF timer.IN THEN
  	timer(IN:=FALSE);
  	timer(IN:=TRUE);
  END_IF;
  narabotka:=0;
  reset:=FALSE;
  END_IF;
END_FUNCTION_BLOCK

CONFIGURATION config1
  VAR_GLOBAL
    systime_s AT %IL0.10.10 : ULINT;
    systime_ns AT %IL0.10.11 : ULINT;
    current_retrieve_us AT %IL0.10.12 : ULINT;
    current_config_us AT %IL0.10.13 : ULINT;
    current_publish_us AT %IL0.10.14 : ULINT;
    current_run_us AT %IL0.10.15 : ULINT;
    max_retrieve_us AT %QL0.10.16 : ULINT;
    max_config_us AT %QL0.10.17 : ULINT;
    max_publish_us AT %QL0.10.18 : ULINT;
    plc_run_number AT %IL0.10.19 : ULINT;
    arAIN_0 : TItemAIN;
    arAIN_1 : TItemAIN;
    arAIN_2 : TItemAIN;
    arAIN_3 : TItemAIN;
    arAIN_4 : TItemAIN;
    arAIN_5 : TItemAIN;
    arAIN_6 : TItemAIN;
    arAIN_7 : TItemAIN;
    arAIN_8 : TItemAIN;
    arAIN_9 : TItemAIN;
    arAIN_10 : TItemAIN;
    arAIN_11 : TItemAIN;
    arAIN_12 : TItemAIN;
    arAIN_13 : TItemAIN;
    arAIN_14 : TItemAIN;
    arAIN_15 : TItemAIN;
    arAIN_16 : TItemAIN;
    arAIN_17 : TItemAIN;
    arAIN_18 : TItemAIN;
    arAIN_19 : TItemAIN;
    arAIN_20 : TItemAIN;
    arAIN_21 : TItemAIN;
    arAIN_22 : TItemAIN;
    arAIN_23 : TItemAIN;
    arAIN_24 : TItemAIN;
    arAIN_25 : TItemAIN;
    arAIN_26 : TItemAIN;
    arAIN_27 : TItemAIN;
    arAIN_28 : TItemAIN;
    arAIN_29 : TItemAIN;
    arAIN_30 : TItemAIN;
    arAIN_31 : TItemAIN;
    arAIN_32 : TItemAIN;
    arAIN_33 : TItemAIN;
    arAIN_34 : TItemAIN;
    arAIN_35 : TItemAIN;
    arAIN_36 : TItemAIN;
    arAIN_37 : TItemAIN;
    arAIN_38 : TItemAIN;
    arAIN_39 : TItemAIN;
    arAIN_40 : TItemAIN;
    arAIN_41 : TItemAIN;
    arAIN_42 : TItemAIN;
    arAIN_43 : TItemAIN;
    arAIN_44 : TItemAIN;
    arAIN_45 : TItemAIN;
    arAIN_46 : TItemAIN;
    arAIN_47 : TItemAIN;
    arAIN_48 : TItemAIN;
    arAIN_49 : TItemAIN;
    arAIN_50 : TItemAIN;
    arAIN_51 : TItemAIN;
    arAIN_52 : TItemAIN;
    arAIN_53 : TItemAIN;
    arAIN_54 : TItemAIN;
    arAIN_55 : TItemAIN;
    arAIN_56 : TItemAIN;
    arAIN_57 : TItemAIN;
    arAIN_58 : TItemAIN;
    arAIN_59 : TItemAIN;
    arAIN_60 : TItemAIN;
    arAIN_61 : TItemAIN;
    arAIN_62 : TItemAIN;
    arAIN_63 : TItemAIN;
    arAIN_64 : TItemAIN;
    arAIN_65 : TItemAIN;
    arAIN_66 : TItemAIN;
    arAIN_67 : TItemAIN;
    arAIN_68 : TItemAIN;
    arAIN_69 : TItemAIN;
    arAIN_70 : TItemAIN;
    arAIN_71 : TItemAIN;
    arAIN_72 : TItemAIN;
    arAIN_73 : TItemAIN;
    arAIN_74 : TItemAIN;
    arAIN_75 : TItemAIN;
    arAIN_76 : TItemAIN;
    arAIN_77 : TItemAIN;
    arAIN_78 : TItemAIN;
    arAIN_79 : TItemAIN;
    arDIN_0 : TItemDIN;
    arDIN_1 : TItemDIN;
    arDIN_2 : TItemDIN;
    arDIN_3 : TItemDIN;
    arDIN_4 : TItemDIN;
    arDIN_5 : TItemDIN;
    arDIN_6 : TItemDIN;
    arDIN_7 : TItemDIN;
    arDIN_8 : TItemDIN;
    arDIN_9 : TItemDIN;
    arDIN_10 : TItemDIN;
    arDIN_11 : TItemDIN;
    arDIN_12 : TItemDIN;
    arDIN_13 : TItemDIN;
    arDIN_14 : TItemDIN;
    arDIN_15 : TItemDIN;
    arDIN_16 : TItemDIN;
    arDIN_17 : TItemDIN;
    arDIN_18 : TItemDIN;
    arDIN_19 : TItemDIN;
    arDIN_20 : TItemDIN;
    arDIN_21 : TItemDIN;
    arAOUT_0 : TDoubleData;
    arAOUT_1 : TDoubleData;
    arDOUT_0 : TWordData;
    arDOUT_1 : TWordData;
    arDOUT_2 : TWordData;
    arDOUT_3 : TWordData;
    arDOUT_4 : TWordData;
    arDOUT_66 : TWordData;
    arERR_0 : TItemDIN;
    arERR_1 : TItemDIN;
    arERR_2 : TItemDIN;
    arERR_3 : TItemDIN;
    arERR_4 : TItemDIN;
    arERR_5 : TItemDIN;
    arERR_6 : TItemDIN;
    arERR_7 : TItemDIN;
    arERR_8 : TItemDIN;
    arERR_9 : TItemDIN;
    arERR_10 : TItemDIN;
    arERR_11 : TItemDIN;
    arERR_12 : TItemDIN;
    arERR_13 : TItemDIN;
    arERR_14 : TItemDIN;
    arERR_15 : TItemDIN;
    arERR_16 : TItemDIN;
    arERR_17 : TItemDIN;
    arERR_18 : TItemDIN;
    arERR_19 : TItemDIN;
    arERR_20 : TItemDIN;
    arERR_21 : TItemDIN;
    arERR_22 : TItemDIN;
    arERR_66 : TItemDIN;
    arRelSt_0 : TItemDIN;
  END_VAR

  RESOURCE resource1 ON PLC
    VAR_GLOBAL CONSTANT
      gMaint_Time : REAL;
    END_VAR
    VAR_GLOBAL
      cur_Cycle : REAL;
      gStart_Tmr : REAL;
    END_VAR
    VAR_GLOBAL CONSTANT
      req_Cycle : REAL := 0.02;
    END_VAR
    VAR_GLOBAL
      gF_T_100mSec : BOOL;
      gT_1Sec : BOOL;
      gF_T_1Sec : BOOL;
      gT_1Min : BOOL;
      gR_T_1Min : BOOL;
      gF_T_1Min : BOOL;
      T_1SEC : REAL;
      del_T : REAL;
      ai : AiConfig;
      di : DiConfig;
      od : DOconfig;
      ao : AOConfig;
      IM : ImConfig;
      protections : ProtectionsConfig;
      algoritms : AlgoritmsConfig;
      algManager : struct_AlgoritmsManager;
      ModeGpa : TYPE_ModeGpa;
      protectManager : struct_ProtectionsManager;
      NotHasRezervNU : BOOL;
      Reset_HasNU : BOOL;
      AlgTimers : struct_AlgTimers;
      AlgQuestions : AlgoritmsQuestions;
      PMcommand : TYPE_CommandsPotectionsManager;
      AI_Aktivnaia_moshchnost_HL AT %QL0.2 : LREAL;
      AI_Aktivnaia_moshchnost_LL AT %QL0.3 : LREAL;
      AI_Aktivnaia_moshchnost_command AT %QW0.1 : UINT;
      AI_Aktivnaia_moshchnost_newHL AT %QL0.4 : LREAL;
      AI_Aktivnaia_moshchnost_newLL AT %QL0.5 : LREAL;
      AI_Aktivnaia_moshchnost_status AT %QD0.6 : UDINT;
      AI_Aktivnaia_moshchnost_value AT %QL0.7 : LREAL;
      AI_Osevoi_sdvig_rotora_nagnetatelia_HA AT %QL0.27 : LREAL;
      AI_Osevoi_sdvig_rotora_nagnetatelia_HL AT %QL0.28 : LREAL;
      AI_Osevoi_sdvig_rotora_nagnetatelia_HW AT %QL0.29 : LREAL;
      AI_Osevoi_sdvig_rotora_nagnetatelia_LA AT %QL0.30 : LREAL;
      AI_Osevoi_sdvig_rotora_nagnetatelia_LL AT %QL0.31 : LREAL;
      AI_Osevoi_sdvig_rotora_nagnetatelia_LW AT %QL0.32 : LREAL;
      AI_Osevoi_sdvig_rotora_nagnetatelia_command AT %QW0.26 : UINT;
      AI_Osevoi_sdvig_rotora_nagnetatelia_newHA AT %QL0.33 : LREAL;
      AI_Osevoi_sdvig_rotora_nagnetatelia_newHL AT %QL0.34 : LREAL;
      AI_Osevoi_sdvig_rotora_nagnetatelia_newHW AT %QL0.35 : LREAL;
      AI_Osevoi_sdvig_rotora_nagnetatelia_newLA AT %QL0.36 : LREAL;
      AI_Osevoi_sdvig_rotora_nagnetatelia_newLL AT %QL0.37 : LREAL;
      AI_Osevoi_sdvig_rotora_nagnetatelia_newLW AT %QL0.38 : LREAL;
      AI_Osevoi_sdvig_rotora_nagnetatelia_status AT %QD0.39 : UDINT;
      AI_Osevoi_sdvig_rotora_nagnetatelia_value AT %QL0.40 : LREAL;
      AI_P_gaza_na_vkhode_nagnetatelia_HL AT %QL0.42 : LREAL;
      AI_P_gaza_na_vkhode_nagnetatelia_LL AT %QL0.43 : LREAL;
      AI_P_gaza_na_vkhode_nagnetatelia_command AT %QW0.41 : UINT;
      AI_P_gaza_na_vkhode_nagnetatelia_newHL AT %QL0.44 : LREAL;
      AI_P_gaza_na_vkhode_nagnetatelia_newLL AT %QL0.45 : LREAL;
      AI_P_gaza_na_vkhode_nagnetatelia_status AT %QD0.46 : UDINT;
      AI_P_gaza_na_vkhode_nagnetatelia_value AT %QL0.47 : LREAL;
      AI_P_gaza_na_vykhode_nagnetatelia_HL AT %QL0.49 : LREAL;
      AI_P_gaza_na_vykhode_nagnetatelia_LL AT %QL0.50 : LREAL;
      AI_P_gaza_na_vykhode_nagnetatelia_command AT %QW0.48 : UINT;
      AI_P_gaza_na_vykhode_nagnetatelia_newHL AT %QL0.51 : LREAL;
      AI_P_gaza_na_vykhode_nagnetatelia_newLL AT %QL0.52 : LREAL;
      AI_P_gaza_na_vykhode_nagnetatelia_status AT %QD0.53 : UDINT;
      AI_P_gaza_na_vykhode_nagnetatelia_value AT %QL0.54 : LREAL;
      AI_P_masla_smazki_nizkoe_HL AT %QL0.56 : LREAL;
      AI_P_masla_smazki_nizkoe_LA AT %QL0.57 : LREAL;
      AI_P_masla_smazki_nizkoe_LL AT %QL0.58 : LREAL;
      AI_P_masla_smazki_nizkoe_LW AT %QL0.59 : LREAL;
      AI_P_masla_smazki_nizkoe_command AT %QW0.55 : UINT;
      AI_P_masla_smazki_nizkoe_newHL AT %QL0.60 : LREAL;
      AI_P_masla_smazki_nizkoe_newLA AT %QL0.61 : LREAL;
      AI_P_masla_smazki_nizkoe_newLL AT %QL0.62 : LREAL;
      AI_P_masla_smazki_nizkoe_newLW AT %QL0.63 : LREAL;
      AI_P_masla_smazki_nizkoe_status AT %QD0.64 : UDINT;
      AI_P_masla_smazki_nizkoe_value AT %QL0.65 : LREAL;
      AI_P_masla_smazki_srednee_posle_nasosov_HL AT %QL0.67 : LREAL;
      AI_P_masla_smazki_srednee_posle_nasosov_LL AT %QL0.68 : LREAL;
      AI_P_masla_smazki_srednee_posle_nasosov_LW AT %QL0.69 : LREAL;
      AI_P_masla_smazki_srednee_posle_nasosov_command AT %QW0.66 : UINT;
      AI_P_masla_smazki_srednee_posle_nasosov_newHL AT %QL0.70 : LREAL;
      AI_P_masla_smazki_srednee_posle_nasosov_newLL AT %QL0.71 : LREAL;
      AI_P_masla_smazki_srednee_posle_nasosov_newLW AT %QL0.72 : LREAL;
      AI_P_masla_smazki_srednee_posle_nasosov_status AT %QD0.73 : UDINT;
      AI_P_masla_smazki_srednee_posle_nasosov_value AT %QL0.74 : LREAL;
      AI_P_masla_uplotneniia_HL AT %QL0.76 : LREAL;
      AI_P_masla_uplotneniia_LL AT %QL0.77 : LREAL;
      AI_P_masla_uplotneniia_command AT %QW0.75 : UINT;
      AI_P_masla_uplotneniia_newHL AT %QL0.78 : LREAL;
      AI_P_masla_uplotneniia_newLL AT %QL0.79 : LREAL;
      AI_P_masla_uplotneniia_status AT %QD0.80 : UDINT;
      AI_P_masla_uplotneniia_value AT %QL0.81 : LREAL;
      AI_Reaktivnaia_moshchnost_HL AT %QL0.83 : LREAL;
      AI_Reaktivnaia_moshchnost_LL AT %QL0.84 : LREAL;
      AI_Reaktivnaia_moshchnost_command AT %QW0.82 : UINT;
      AI_Reaktivnaia_moshchnost_newHL AT %QL0.85 : LREAL;
      AI_Reaktivnaia_moshchnost_newLL AT %QL0.86 : LREAL;
      AI_Reaktivnaia_moshchnost_status AT %QD0.87 : UDINT;
      AI_Reaktivnaia_moshchnost_value AT %QL0.88 : LREAL;
      AI_T_aktivnogo_zheleza_statora_1_k_HL AT %QL0.90 : LREAL;
      AI_T_aktivnogo_zheleza_statora_1_k_LL AT %QL0.91 : LREAL;
      AI_T_aktivnogo_zheleza_statora_1_k_command AT %QW0.89 : UINT;
      AI_T_aktivnogo_zheleza_statora_1_k_newHL AT %QL0.92 : LREAL;
      AI_T_aktivnogo_zheleza_statora_1_k_newLL AT %QL0.93 : LREAL;
      AI_T_aktivnogo_zheleza_statora_1_k_status AT %QD0.94 : UDINT;
      AI_T_aktivnogo_zheleza_statora_1_k_value AT %QL0.95 : LREAL;
      AI_T_aktivnogo_zheleza_statora_2_k_HL AT %QL0.97 : LREAL;
      AI_T_aktivnogo_zheleza_statora_2_k_LL AT %QL0.98 : LREAL;
      AI_T_aktivnogo_zheleza_statora_2_k_command AT %QW0.96 : UINT;
      AI_T_aktivnogo_zheleza_statora_2_k_newHL AT %QL0.99 : LREAL;
      AI_T_aktivnogo_zheleza_statora_2_k_newLL AT %QL0.100 : LREAL;
      AI_T_aktivnogo_zheleza_statora_2_k_status AT %QD0.101 : UDINT;
      AI_T_aktivnogo_zheleza_statora_2_k_value AT %QL0.102 : LREAL;
      AI_T_aktivnogo_zheleza_statora_3_k_HL AT %QL0.104 : LREAL;
      AI_T_aktivnogo_zheleza_statora_3_k_LL AT %QL0.105 : LREAL;
      AI_T_aktivnogo_zheleza_statora_3_k_command AT %QW0.103 : UINT;
      AI_T_aktivnogo_zheleza_statora_3_k_newHL AT %QL0.106 : LREAL;
      AI_T_aktivnogo_zheleza_statora_3_k_newLL AT %QL0.107 : LREAL;
      AI_T_aktivnogo_zheleza_statora_3_k_status AT %QD0.108 : UDINT;
      AI_T_aktivnogo_zheleza_statora_3_k_value AT %QL0.109 : LREAL;
      AI_T_clodAir_dvigatelia_t1_HL AT %QL0.111 : LREAL;
      AI_T_clodAir_dvigatelia_t1_LL AT %QL0.112 : LREAL;
      AI_T_clodAir_dvigatelia_t1_command AT %QW0.110 : UINT;
      AI_T_clodAir_dvigatelia_t1_newHL AT %QL0.113 : LREAL;
      AI_T_clodAir_dvigatelia_t1_newLL AT %QL0.114 : LREAL;
      AI_T_clodAir_dvigatelia_t1_status AT %QD0.115 : UDINT;
      AI_T_clodAir_dvigatelia_t1_value AT %QL0.116 : LREAL;
      AI_T_gaz_in_nagnetatelia_HL AT %QL0.118 : LREAL;
      AI_T_gaz_in_nagnetatelia_LL AT %QL0.119 : LREAL;
      AI_T_gaz_in_nagnetatelia_command AT %QW0.117 : UINT;
      AI_T_gaz_in_nagnetatelia_newHL AT %QL0.120 : LREAL;
      AI_T_gaz_in_nagnetatelia_newLL AT %QL0.121 : LREAL;
      AI_T_gaz_in_nagnetatelia_status AT %QD0.122 : UDINT;
      AI_T_gaz_in_nagnetatelia_value AT %QL0.123 : LREAL;
      AI_T_gaz_out_nagnetatelia_HA AT %QL0.125 : LREAL;
      AI_T_gaz_out_nagnetatelia_HL AT %QL0.126 : LREAL;
      AI_T_gaz_out_nagnetatelia_HW AT %QL0.127 : LREAL;
      AI_T_gaz_out_nagnetatelia_LL AT %QL0.128 : LREAL;
      AI_T_gaz_out_nagnetatelia_command AT %QW0.124 : UINT;
      AI_T_gaz_out_nagnetatelia_newHA AT %QL0.129 : LREAL;
      AI_T_gaz_out_nagnetatelia_newHL AT %QL0.130 : LREAL;
      AI_T_gaz_out_nagnetatelia_newHW AT %QL0.131 : LREAL;
      AI_T_gaz_out_nagnetatelia_newLL AT %QL0.132 : LREAL;
      AI_T_gaz_out_nagnetatelia_status AT %QD0.133 : UDINT;
      AI_T_gaz_out_nagnetatelia_value AT %QL0.134 : LREAL;
      AI_T_hotAir_dvigatelia_t1_HL AT %QL0.136 : LREAL;
      AI_T_hotAir_dvigatelia_t1_LL AT %QL0.137 : LREAL;
      AI_T_hotAir_dvigatelia_t1_command AT %QW0.135 : UINT;
      AI_T_hotAir_dvigatelia_t1_newHL AT %QL0.138 : LREAL;
      AI_T_hotAir_dvigatelia_t1_newLL AT %QL0.139 : LREAL;
      AI_T_hotAir_dvigatelia_t1_status AT %QD0.140 : UDINT;
      AI_T_hotAir_dvigatelia_t1_value AT %QL0.141 : LREAL;
      AI_T_masla_do_AVOM_HL AT %QL0.143 : LREAL;
      AI_T_masla_do_AVOM_LL AT %QL0.144 : LREAL;
      AI_T_masla_do_AVOM_command AT %QW0.142 : UINT;
      AI_T_masla_do_AVOM_newHL AT %QL0.145 : LREAL;
      AI_T_masla_do_AVOM_newLL AT %QL0.146 : LREAL;
      AI_T_masla_do_AVOM_status AT %QD0.147 : UDINT;
      AI_T_masla_do_AVOM_value AT %QL0.148 : LREAL;
      AI_T_masla_na_slive_perednego_opornogo_podshipnika_dvigatelia_HL AT %QL0.150 : LREAL;
      AI_T_masla_na_slive_perednego_opornogo_podshipnika_dvigatelia_LL AT %QL0.151 : LREAL;
      AI_T_masla_na_slive_perednego_opornogo_podshipnika_dvigatelia_command AT %QW0.149 : UINT;
      AI_T_masla_na_slive_perednego_opornogo_podshipnika_dvigatelia_newHL AT %QL0.152 : LREAL;
      AI_T_masla_na_slive_perednego_opornogo_podshipnika_dvigatelia_newLL AT %QL0.153 : LREAL;
      AI_T_masla_na_slive_perednego_opornogo_podshipnika_dvigatelia_status AT %QD0.154 : UDINT;
      AI_T_masla_na_slive_perednego_opornogo_podshipnika_dvigatelia_value AT %QL0.155 : LREAL;
      AI_T_masla_na_slive_zadnego_opornogo_podshipnika_dvigatelia_HL AT %QL0.157 : LREAL;
      AI_T_masla_na_slive_zadnego_opornogo_podshipnika_dvigatelia_LL AT %QL0.158 : LREAL;
      AI_T_masla_na_slive_zadnego_opornogo_podshipnika_dvigatelia_command AT %QW0.156 : UINT;
      AI_T_masla_na_slive_zadnego_opornogo_podshipnika_dvigatelia_newHL AT %QL0.159 : LREAL;
      AI_T_masla_na_slive_zadnego_opornogo_podshipnika_dvigatelia_newLL AT %QL0.160 : LREAL;
      AI_T_masla_na_slive_zadnego_opornogo_podshipnika_dvigatelia_status AT %QD0.161 : UDINT;
      AI_T_masla_na_slive_zadnego_opornogo_podshipnika_dvigatelia_value AT %QL0.162 : LREAL;
      AI_T_masla_posle_AVOM_HL AT %QL0.164 : LREAL;
      AI_T_masla_posle_AVOM_LL AT %QL0.165 : LREAL;
      AI_T_masla_posle_AVOM_command AT %QW0.163 : UINT;
      AI_T_masla_posle_AVOM_newHL AT %QL0.166 : LREAL;
      AI_T_masla_posle_AVOM_newLL AT %QL0.167 : LREAL;
      AI_T_masla_posle_AVOM_status AT %QD0.168 : UDINT;
      AI_T_masla_posle_AVOM_value AT %QL0.169 : LREAL;
      AI_T_masla_v_maslobake_HL AT %QL0.171 : LREAL;
      AI_T_masla_v_maslobake_HW AT %QL0.172 : LREAL;
      AI_T_masla_v_maslobake_LL AT %QL0.173 : LREAL;
      AI_T_masla_v_maslobake_LW AT %QL0.174 : LREAL;
      AI_T_masla_v_maslobake_command AT %QW0.170 : UINT;
      AI_T_masla_v_maslobake_newHL AT %QL0.175 : LREAL;
      AI_T_masla_v_maslobake_newHW AT %QL0.176 : LREAL;
      AI_T_masla_v_maslobake_newLL AT %QL0.177 : LREAL;
      AI_T_masla_v_maslobake_newLW AT %QL0.178 : LREAL;
      AI_T_masla_v_maslobake_status AT %QD0.179 : UDINT;
      AI_T_masla_v_maslobake_value AT %QL0.180 : LREAL;
      AI_T_obmotki_fazy_1_k_HL AT %QL0.182 : LREAL;
      AI_T_obmotki_fazy_1_k_LL AT %QL0.183 : LREAL;
      AI_T_obmotki_fazy_1_k_command AT %QW0.181 : UINT;
      AI_T_obmotki_fazy_1_k_newHL AT %QL0.184 : LREAL;
      AI_T_obmotki_fazy_1_k_newLL AT %QL0.185 : LREAL;
      AI_T_obmotki_fazy_1_k_status AT %QD0.186 : UDINT;
      AI_T_obmotki_fazy_1_k_value AT %QL0.187 : LREAL;
      AI_T_obmotki_fazy_2_k_HL AT %QL0.189 : LREAL;
      AI_T_obmotki_fazy_2_k_LL AT %QL0.190 : LREAL;
      AI_T_obmotki_fazy_2_k_command AT %QW0.188 : UINT;
      AI_T_obmotki_fazy_2_k_newHL AT %QL0.191 : LREAL;
      AI_T_obmotki_fazy_2_k_newLL AT %QL0.192 : LREAL;
      AI_T_obmotki_fazy_2_k_status AT %QD0.193 : UDINT;
      AI_T_obmotki_fazy_2_k_value AT %QL0.194 : LREAL;
      AI_T_obmotki_fazy_3_k_HL AT %QL0.196 : LREAL;
      AI_T_obmotki_fazy_3_k_LL AT %QL0.197 : LREAL;
      AI_T_obmotki_fazy_3_k_command AT %QW0.195 : UINT;
      AI_T_obmotki_fazy_3_k_newHL AT %QL0.198 : LREAL;
      AI_T_obmotki_fazy_3_k_newLL AT %QL0.199 : LREAL;
      AI_T_obmotki_fazy_3_k_status AT %QD0.200 : UDINT;
      AI_T_obmotki_fazy_3_k_value AT %QL0.201 : LREAL;
      AI_T_oporno_upornogo_podshipnika_nagnetatelia_t4_HA AT %QL0.203 : LREAL;
      AI_T_oporno_upornogo_podshipnika_nagnetatelia_t4_HL AT %QL0.204 : LREAL;
      AI_T_oporno_upornogo_podshipnika_nagnetatelia_t4_HW AT %QL0.205 : LREAL;
      AI_T_oporno_upornogo_podshipnika_nagnetatelia_t4_LL AT %QL0.206 : LREAL;
      AI_T_oporno_upornogo_podshipnika_nagnetatelia_t4_command AT %QW0.202 : UINT;
      AI_T_oporno_upornogo_podshipnika_nagnetatelia_t4_newHA AT %QL0.207 : LREAL;
      AI_T_oporno_upornogo_podshipnika_nagnetatelia_t4_newHL AT %QL0.208 : LREAL;
      AI_T_oporno_upornogo_podshipnika_nagnetatelia_t4_newHW AT %QL0.209 : LREAL;
      AI_T_oporno_upornogo_podshipnika_nagnetatelia_t4_newLL AT %QL0.210 : LREAL;
      AI_T_oporno_upornogo_podshipnika_nagnetatelia_t4_status AT %QD0.211 : UDINT;
      AI_T_oporno_upornogo_podshipnika_nagnetatelia_t4_value AT %QL0.212 : LREAL;
      AI_T_opornogo_podshipnika_nagnetatelia_t1_HA AT %QL0.214 : LREAL;
      AI_T_opornogo_podshipnika_nagnetatelia_t1_HL AT %QL0.215 : LREAL;
      AI_T_opornogo_podshipnika_nagnetatelia_t1_HW AT %QL0.216 : LREAL;
      AI_T_opornogo_podshipnika_nagnetatelia_t1_LL AT %QL0.217 : LREAL;
      AI_T_opornogo_podshipnika_nagnetatelia_t1_command AT %QW0.213 : UINT;
      AI_T_opornogo_podshipnika_nagnetatelia_t1_newHA AT %QL0.218 : LREAL;
      AI_T_opornogo_podshipnika_nagnetatelia_t1_newHL AT %QL0.219 : LREAL;
      AI_T_opornogo_podshipnika_nagnetatelia_t1_newHW AT %QL0.220 : LREAL;
      AI_T_opornogo_podshipnika_nagnetatelia_t1_newLL AT %QL0.221 : LREAL;
      AI_T_opornogo_podshipnika_nagnetatelia_t1_status AT %QD0.222 : UDINT;
      AI_T_opornogo_podshipnika_nagnetatelia_t1_value AT %QL0.223 : LREAL;
      AI_T_opornogo_podshipnika_nagnetatelia_t2_HA AT %QL0.225 : LREAL;
      AI_T_opornogo_podshipnika_nagnetatelia_t2_HL AT %QL0.226 : LREAL;
      AI_T_opornogo_podshipnika_nagnetatelia_t2_HW AT %QL0.227 : LREAL;
      AI_T_opornogo_podshipnika_nagnetatelia_t2_LL AT %QL0.228 : LREAL;
      AI_T_opornogo_podshipnika_nagnetatelia_t2_command AT %QW0.224 : UINT;
      AI_T_opornogo_podshipnika_nagnetatelia_t2_newHA AT %QL0.229 : LREAL;
      AI_T_opornogo_podshipnika_nagnetatelia_t2_newHL AT %QL0.230 : LREAL;
      AI_T_opornogo_podshipnika_nagnetatelia_t2_newHW AT %QL0.231 : LREAL;
      AI_T_opornogo_podshipnika_nagnetatelia_t2_newLL AT %QL0.232 : LREAL;
      AI_T_opornogo_podshipnika_nagnetatelia_t2_status AT %QD0.233 : UDINT;
      AI_T_opornogo_podshipnika_nagnetatelia_t2_value AT %QL0.234 : LREAL;
      AI_T_opornogo_podshipnika_nagnetatelia_t3_HA AT %QL0.236 : LREAL;
      AI_T_opornogo_podshipnika_nagnetatelia_t3_HL AT %QL0.237 : LREAL;
      AI_T_opornogo_podshipnika_nagnetatelia_t3_HW AT %QL0.238 : LREAL;
      AI_T_opornogo_podshipnika_nagnetatelia_t3_LL AT %QL0.239 : LREAL;
      AI_T_opornogo_podshipnika_nagnetatelia_t3_command AT %QW0.235 : UINT;
      AI_T_opornogo_podshipnika_nagnetatelia_t3_newHA AT %QL0.240 : LREAL;
      AI_T_opornogo_podshipnika_nagnetatelia_t3_newHL AT %QL0.241 : LREAL;
      AI_T_opornogo_podshipnika_nagnetatelia_t3_newHW AT %QL0.242 : LREAL;
      AI_T_opornogo_podshipnika_nagnetatelia_t3_newLL AT %QL0.243 : LREAL;
      AI_T_opornogo_podshipnika_nagnetatelia_t3_status AT %QD0.244 : UDINT;
      AI_T_opornogo_podshipnika_nagnetatelia_t3_value AT %QL0.245 : LREAL;
      AI_T_perednego_opornogo_podshipnika_dvigatelia_t1_HA AT %QL0.247 : LREAL;
      AI_T_perednego_opornogo_podshipnika_dvigatelia_t1_HL AT %QL0.248 : LREAL;
      AI_T_perednego_opornogo_podshipnika_dvigatelia_t1_HW AT %QL0.249 : LREAL;
      AI_T_perednego_opornogo_podshipnika_dvigatelia_t1_LL AT %QL0.250 : LREAL;
      AI_T_perednego_opornogo_podshipnika_dvigatelia_t1_command AT %QW0.246 : UINT;
      AI_T_perednego_opornogo_podshipnika_dvigatelia_t1_newHA AT %QL0.251 : LREAL;
      AI_T_perednego_opornogo_podshipnika_dvigatelia_t1_newHL AT %QL0.252 : LREAL;
      AI_T_perednego_opornogo_podshipnika_dvigatelia_t1_newHW AT %QL0.253 : LREAL;
      AI_T_perednego_opornogo_podshipnika_dvigatelia_t1_newLL AT %QL0.254 : LREAL;
      AI_T_perednego_opornogo_podshipnika_dvigatelia_t1_status AT %QD0.255 : UDINT;
      AI_T_perednego_opornogo_podshipnika_dvigatelia_t1_value AT %QL0.256 : LREAL;
      AI_T_podshipnika_reduktora_t1_HA AT %QL0.258 : LREAL;
      AI_T_podshipnika_reduktora_t1_HL AT %QL0.259 : LREAL;
      AI_T_podshipnika_reduktora_t1_HW AT %QL0.260 : LREAL;
      AI_T_podshipnika_reduktora_t1_LL AT %QL0.261 : LREAL;
      AI_T_podshipnika_reduktora_t1_command AT %QW0.257 : UINT;
      AI_T_podshipnika_reduktora_t1_newHA AT %QL0.262 : LREAL;
      AI_T_podshipnika_reduktora_t1_newHL AT %QL0.263 : LREAL;
      AI_T_podshipnika_reduktora_t1_newHW AT %QL0.264 : LREAL;
      AI_T_podshipnika_reduktora_t1_newLL AT %QL0.265 : LREAL;
      AI_T_podshipnika_reduktora_t1_status AT %QD0.266 : UDINT;
      AI_T_podshipnika_reduktora_t1_value AT %QL0.267 : LREAL;
      AI_T_podshipnika_reduktora_t2_HA AT %QL0.269 : LREAL;
      AI_T_podshipnika_reduktora_t2_HL AT %QL0.270 : LREAL;
      AI_T_podshipnika_reduktora_t2_HW AT %QL0.271 : LREAL;
      AI_T_podshipnika_reduktora_t2_LL AT %QL0.272 : LREAL;
      AI_T_podshipnika_reduktora_t2_command AT %QW0.268 : UINT;
      AI_T_podshipnika_reduktora_t2_newHA AT %QL0.273 : LREAL;
      AI_T_podshipnika_reduktora_t2_newHL AT %QL0.274 : LREAL;
      AI_T_podshipnika_reduktora_t2_newHW AT %QL0.275 : LREAL;
      AI_T_podshipnika_reduktora_t2_newLL AT %QL0.276 : LREAL;
      AI_T_podshipnika_reduktora_t2_status AT %QD0.277 : UDINT;
      AI_T_podshipnika_reduktora_t2_value AT %QL0.278 : LREAL;
      AI_T_podshipnika_reduktora_t3_HA AT %QL0.280 : LREAL;
      AI_T_podshipnika_reduktora_t3_HL AT %QL0.281 : LREAL;
      AI_T_podshipnika_reduktora_t3_HW AT %QL0.282 : LREAL;
      AI_T_podshipnika_reduktora_t3_LL AT %QL0.283 : LREAL;
      AI_T_podshipnika_reduktora_t3_command AT %QW0.279 : UINT;
      AI_T_podshipnika_reduktora_t3_newHA AT %QL0.284 : LREAL;
      AI_T_podshipnika_reduktora_t3_newHL AT %QL0.285 : LREAL;
      AI_T_podshipnika_reduktora_t3_newHW AT %QL0.286 : LREAL;
      AI_T_podshipnika_reduktora_t3_newLL AT %QL0.287 : LREAL;
      AI_T_podshipnika_reduktora_t3_status AT %QD0.288 : UDINT;
      AI_T_podshipnika_reduktora_t3_value AT %QL0.289 : LREAL;
      AI_T_podshipnika_reduktora_t4_HA AT %QL0.291 : LREAL;
      AI_T_podshipnika_reduktora_t4_HL AT %QL0.292 : LREAL;
      AI_T_podshipnika_reduktora_t4_HW AT %QL0.293 : LREAL;
      AI_T_podshipnika_reduktora_t4_LL AT %QL0.294 : LREAL;
      AI_T_podshipnika_reduktora_t4_command AT %QW0.290 : UINT;
      AI_T_podshipnika_reduktora_t4_newHA AT %QL0.295 : LREAL;
      AI_T_podshipnika_reduktora_t4_newHL AT %QL0.296 : LREAL;
      AI_T_podshipnika_reduktora_t4_newHW AT %QL0.297 : LREAL;
      AI_T_podshipnika_reduktora_t4_newLL AT %QL0.298 : LREAL;
      AI_T_podshipnika_reduktora_t4_status AT %QD0.299 : UDINT;
      AI_T_podshipnika_reduktora_t4_value AT %QL0.300 : LREAL;
      AI_T_zadnego_opornogo_podshipnika_dvigatelia_t2_HA AT %QL0.302 : LREAL;
      AI_T_zadnego_opornogo_podshipnika_dvigatelia_t2_HL AT %QL0.303 : LREAL;
      AI_T_zadnego_opornogo_podshipnika_dvigatelia_t2_HW AT %QL0.304 : LREAL;
      AI_T_zadnego_opornogo_podshipnika_dvigatelia_t2_LL AT %QL0.305 : LREAL;
      AI_T_zadnego_opornogo_podshipnika_dvigatelia_t2_command AT %QW0.301 : UINT;
      AI_T_zadnego_opornogo_podshipnika_dvigatelia_t2_newHA AT %QL0.306 : LREAL;
      AI_T_zadnego_opornogo_podshipnika_dvigatelia_t2_newHL AT %QL0.307 : LREAL;
      AI_T_zadnego_opornogo_podshipnika_dvigatelia_t2_newHW AT %QL0.308 : LREAL;
      AI_T_zadnego_opornogo_podshipnika_dvigatelia_t2_newLL AT %QL0.309 : LREAL;
      AI_T_zadnego_opornogo_podshipnika_dvigatelia_t2_status AT %QD0.310 : UDINT;
      AI_T_zadnego_opornogo_podshipnika_dvigatelia_t2_value AT %QL0.311 : LREAL;
      AI_Tok_statora_elektrodvigatelia_HL AT %QL0.313 : LREAL;
      AI_Tok_statora_elektrodvigatelia_LL AT %QL0.314 : LREAL;
      AI_Tok_statora_elektrodvigatelia_command AT %QW0.312 : UINT;
      AI_Tok_statora_elektrodvigatelia_newHL AT %QL0.315 : LREAL;
      AI_Tok_statora_elektrodvigatelia_newLL AT %QL0.316 : LREAL;
      AI_Tok_statora_elektrodvigatelia_status AT %QD0.317 : UDINT;
      AI_Tok_statora_elektrodvigatelia_value AT %QL0.318 : LREAL;
      AI_Tok_vozbuzhdeniia_vozbuditelia_HL AT %QL0.320 : LREAL;
      AI_Tok_vozbuzhdeniia_vozbuditelia_LL AT %QL0.321 : LREAL;
      AI_Tok_vozbuzhdeniia_vozbuditelia_command AT %QW0.319 : UINT;
      AI_Tok_vozbuzhdeniia_vozbuditelia_newHL AT %QL0.322 : LREAL;
      AI_Tok_vozbuzhdeniia_vozbuditelia_newLL AT %QL0.323 : LREAL;
      AI_Tok_vozbuzhdeniia_vozbuditelia_status AT %QD0.324 : UDINT;
      AI_Tok_vozbuzhdeniia_vozbuditelia_value AT %QL0.325 : LREAL;
      AI_Uroven_masla_v_maslobake_HL AT %QL0.327 : LREAL;
      AI_Uroven_masla_v_maslobake_HW AT %QL0.328 : LREAL;
      AI_Uroven_masla_v_maslobake_LA AT %QL0.329 : LREAL;
      AI_Uroven_masla_v_maslobake_LL AT %QL0.330 : LREAL;
      AI_Uroven_masla_v_maslobake_LW AT %QL0.331 : LREAL;
      AI_Uroven_masla_v_maslobake_command AT %QW0.326 : UINT;
      AI_Uroven_masla_v_maslobake_newHL AT %QL0.332 : LREAL;
      AI_Uroven_masla_v_maslobake_newHW AT %QL0.333 : LREAL;
      AI_Uroven_masla_v_maslobake_newLA AT %QL0.334 : LREAL;
      AI_Uroven_masla_v_maslobake_newLL AT %QL0.335 : LREAL;
      AI_Uroven_masla_v_maslobake_newLW AT %QL0.336 : LREAL;
      AI_Uroven_masla_v_maslobake_status AT %QD0.337 : UDINT;
      AI_Uroven_masla_v_maslobake_value AT %QL0.338 : LREAL;
      AI_Vibratciia_STD_t1_HA AT %QL0.384 : LREAL;
      AI_Vibratciia_STD_t1_HL AT %QL0.385 : LREAL;
      AI_Vibratciia_STD_t1_HW AT %QL0.386 : LREAL;
      AI_Vibratciia_STD_t1_LL AT %QL0.387 : LREAL;
      AI_Vibratciia_STD_t1_command AT %QW0.383 : UINT;
      AI_Vibratciia_STD_t1_newHA AT %QL0.388 : LREAL;
      AI_Vibratciia_STD_t1_newHL AT %QL0.389 : LREAL;
      AI_Vibratciia_STD_t1_newHW AT %QL0.390 : LREAL;
      AI_Vibratciia_STD_t1_newLL AT %QL0.391 : LREAL;
      AI_Vibratciia_STD_t1_status AT %QD0.392 : UDINT;
      AI_Vibratciia_STD_t1_value AT %QL0.393 : LREAL;
      AI_Vibratciia_STD_t2_HA AT %QL0.395 : LREAL;
      AI_Vibratciia_STD_t2_HL AT %QL0.396 : LREAL;
      AI_Vibratciia_STD_t2_HW AT %QL0.397 : LREAL;
      AI_Vibratciia_STD_t2_LL AT %QL0.398 : LREAL;
      AI_Vibratciia_STD_t2_command AT %QW0.394 : UINT;
      AI_Vibratciia_STD_t2_newHA AT %QL0.399 : LREAL;
      AI_Vibratciia_STD_t2_newHL AT %QL0.400 : LREAL;
      AI_Vibratciia_STD_t2_newHW AT %QL0.401 : LREAL;
      AI_Vibratciia_STD_t2_newLL AT %QL0.402 : LREAL;
      AI_Vibratciia_STD_t2_status AT %QD0.403 : UDINT;
      AI_Vibratciia_STD_t2_value AT %QL0.404 : LREAL;
      AI_Vibratciia_rotora_nagnetatelia_t1_HA AT %QL0.340 : LREAL;
      AI_Vibratciia_rotora_nagnetatelia_t1_HL AT %QL0.341 : LREAL;
      AI_Vibratciia_rotora_nagnetatelia_t1_HW AT %QL0.342 : LREAL;
      AI_Vibratciia_rotora_nagnetatelia_t1_LL AT %QL0.343 : LREAL;
      AI_Vibratciia_rotora_nagnetatelia_t1_command AT %QW0.339 : UINT;
      AI_Vibratciia_rotora_nagnetatelia_t1_newHA AT %QL0.344 : LREAL;
      AI_Vibratciia_rotora_nagnetatelia_t1_newHL AT %QL0.345 : LREAL;
      AI_Vibratciia_rotora_nagnetatelia_t1_newHW AT %QL0.346 : LREAL;
      AI_Vibratciia_rotora_nagnetatelia_t1_newLL AT %QL0.347 : LREAL;
      AI_Vibratciia_rotora_nagnetatelia_t1_status AT %QD0.348 : UDINT;
      AI_Vibratciia_rotora_nagnetatelia_t1_value AT %QL0.349 : LREAL;
      AI_Vibratciia_rotora_nagnetatelia_t2_HA AT %QL0.351 : LREAL;
      AI_Vibratciia_rotora_nagnetatelia_t2_HL AT %QL0.352 : LREAL;
      AI_Vibratciia_rotora_nagnetatelia_t2_HW AT %QL0.353 : LREAL;
      AI_Vibratciia_rotora_nagnetatelia_t2_LL AT %QL0.354 : LREAL;
      AI_Vibratciia_rotora_nagnetatelia_t2_command AT %QW0.350 : UINT;
      AI_Vibratciia_rotora_nagnetatelia_t2_newHA AT %QL0.355 : LREAL;
      AI_Vibratciia_rotora_nagnetatelia_t2_newHL AT %QL0.356 : LREAL;
      AI_Vibratciia_rotora_nagnetatelia_t2_newHW AT %QL0.357 : LREAL;
      AI_Vibratciia_rotora_nagnetatelia_t2_newLL AT %QL0.358 : LREAL;
      AI_Vibratciia_rotora_nagnetatelia_t2_status AT %QD0.359 : UDINT;
      AI_Vibratciia_rotora_nagnetatelia_t2_value AT %QL0.360 : LREAL;
      AI_Vibratciia_rotora_nagnetatelia_t3_HA AT %QL0.362 : LREAL;
      AI_Vibratciia_rotora_nagnetatelia_t3_HL AT %QL0.363 : LREAL;
      AI_Vibratciia_rotora_nagnetatelia_t3_HW AT %QL0.364 : LREAL;
      AI_Vibratciia_rotora_nagnetatelia_t3_LL AT %QL0.365 : LREAL;
      AI_Vibratciia_rotora_nagnetatelia_t3_command AT %QW0.361 : UINT;
      AI_Vibratciia_rotora_nagnetatelia_t3_newHA AT %QL0.366 : LREAL;
      AI_Vibratciia_rotora_nagnetatelia_t3_newHL AT %QL0.367 : LREAL;
      AI_Vibratciia_rotora_nagnetatelia_t3_newHW AT %QL0.368 : LREAL;
      AI_Vibratciia_rotora_nagnetatelia_t3_newLL AT %QL0.369 : LREAL;
      AI_Vibratciia_rotora_nagnetatelia_t3_status AT %QD0.370 : UDINT;
      AI_Vibratciia_rotora_nagnetatelia_t3_value AT %QL0.371 : LREAL;
      AI_Vibratciia_rotora_nagnetatelia_t4_HA AT %QL0.373 : LREAL;
      AI_Vibratciia_rotora_nagnetatelia_t4_HL AT %QL0.374 : LREAL;
      AI_Vibratciia_rotora_nagnetatelia_t4_HW AT %QL0.375 : LREAL;
      AI_Vibratciia_rotora_nagnetatelia_t4_LL AT %QL0.376 : LREAL;
      AI_Vibratciia_rotora_nagnetatelia_t4_command AT %QW0.372 : UINT;
      AI_Vibratciia_rotora_nagnetatelia_t4_newHA AT %QL0.377 : LREAL;
      AI_Vibratciia_rotora_nagnetatelia_t4_newHL AT %QL0.378 : LREAL;
      AI_Vibratciia_rotora_nagnetatelia_t4_newHW AT %QL0.379 : LREAL;
      AI_Vibratciia_rotora_nagnetatelia_t4_newLL AT %QL0.380 : LREAL;
      AI_Vibratciia_rotora_nagnetatelia_t4_status AT %QD0.381 : UDINT;
      AI_Vibratciia_rotora_nagnetatelia_t4_value AT %QL0.382 : LREAL;
      AI_VoltageSHU_osnovnoi_vvod_HL AT %QL0.406 : LREAL;
      AI_VoltageSHU_osnovnoi_vvod_HW AT %QL0.407 : LREAL;
      AI_VoltageSHU_osnovnoi_vvod_LL AT %QL0.408 : LREAL;
      AI_VoltageSHU_osnovnoi_vvod_LW AT %QL0.409 : LREAL;
      AI_VoltageSHU_osnovnoi_vvod_command AT %QW0.405 : UINT;
      AI_VoltageSHU_osnovnoi_vvod_newHL AT %QL0.410 : LREAL;
      AI_VoltageSHU_osnovnoi_vvod_newHW AT %QL0.411 : LREAL;
      AI_VoltageSHU_osnovnoi_vvod_newLL AT %QL0.412 : LREAL;
      AI_VoltageSHU_osnovnoi_vvod_newLW AT %QL0.413 : LREAL;
      AI_VoltageSHU_osnovnoi_vvod_status AT %QD0.414 : UDINT;
      AI_VoltageSHU_osnovnoi_vvod_value AT %QL0.415 : LREAL;
      AI_VoltageSHU_rezervnyi_vvod_HL AT %QL0.417 : LREAL;
      AI_VoltageSHU_rezervnyi_vvod_HW AT %QL0.418 : LREAL;
      AI_VoltageSHU_rezervnyi_vvod_LL AT %QL0.419 : LREAL;
      AI_VoltageSHU_rezervnyi_vvod_LW AT %QL0.420 : LREAL;
      AI_VoltageSHU_rezervnyi_vvod_command AT %QW0.416 : UINT;
      AI_VoltageSHU_rezervnyi_vvod_newHL AT %QL0.421 : LREAL;
      AI_VoltageSHU_rezervnyi_vvod_newHW AT %QL0.422 : LREAL;
      AI_VoltageSHU_rezervnyi_vvod_newLL AT %QL0.423 : LREAL;
      AI_VoltageSHU_rezervnyi_vvod_newLW AT %QL0.424 : LREAL;
      AI_VoltageSHU_rezervnyi_vvod_status AT %QD0.425 : UDINT;
      AI_VoltageSHU_rezervnyi_vvod_value AT %QL0.426 : LREAL;
      AI_dP_gaza_na_konfuzore_nagnetatelia_HL AT %QL0.9 : LREAL;
      AI_dP_gaza_na_konfuzore_nagnetatelia_LL AT %QL0.10 : LREAL;
      AI_dP_gaza_na_konfuzore_nagnetatelia_command AT %QW0.8 : UINT;
      AI_dP_gaza_na_konfuzore_nagnetatelia_newHL AT %QL0.11 : LREAL;
      AI_dP_gaza_na_konfuzore_nagnetatelia_newLL AT %QL0.12 : LREAL;
      AI_dP_gaza_na_konfuzore_nagnetatelia_status AT %QD0.13 : UDINT;
      AI_dP_gaza_na_konfuzore_nagnetatelia_value AT %QL0.14 : LREAL;
      AI_dPmaslo_gaz_HL AT %QL0.16 : LREAL;
      AI_dPmaslo_gaz_LA AT %QL0.17 : LREAL;
      AI_dPmaslo_gaz_LL AT %QL0.18 : LREAL;
      AI_dPmaslo_gaz_LW AT %QL0.19 : LREAL;
      AI_dPmaslo_gaz_command AT %QW0.15 : UINT;
      AI_dPmaslo_gaz_newHL AT %QL0.20 : LREAL;
      AI_dPmaslo_gaz_newLA AT %QL0.21 : LREAL;
      AI_dPmaslo_gaz_newLL AT %QL0.22 : LREAL;
      AI_dPmaslo_gaz_newLW AT %QL0.23 : LREAL;
      AI_dPmaslo_gaz_status AT %QD0.24 : UDINT;
      AI_dPmaslo_gaz_value AT %QL0.25 : LREAL;
      IM_SingleSignals_DverShkafaOtkryta_status AT %QD0.456 : UDINT;
      IM_SingleSignals_KZ_10kv_status AT %QD0.457 : UDINT;
      IM_SingleSignals_NOGPA_knopkaSHU_status AT %QD0.453 : UDINT;
      IM_SingleSignals_NS_G10_G11_status AT %QD0.481 : UDINT;
      IM_SingleSignals_NS_G13_G14_status AT %QD0.482 : UDINT;
      IM_SingleSignals_NS_G15_G16_status AT %QD0.483 : UDINT;
      IM_SingleSignals_NS_G17_status AT %QD0.484 : UDINT;
      IM_SingleSignals_NS_G18_G19_status AT %QD0.485 : UDINT;
      IM_SingleSignals_NS_G1_G2_status AT %QD0.477 : UDINT;
      IM_SingleSignals_NS_G3_G4_status AT %QD0.478 : UDINT;
      IM_SingleSignals_NS_G5_G6_status AT %QD0.479 : UDINT;
      IM_SingleSignals_NS_G7_G8_status AT %QD0.480 : UDINT;
      IM_SingleSignals_OsevoiSdvig_levo_status AT %QD0.458 : UDINT;
      IM_SingleSignals_OsevoiSdvig_pravo_status AT %QD0.459 : UDINT;
      IM_SingleSignals_P_oil_low_status AT %QD0.455 : UDINT;
      IM_SingleSignals_QF10_QF11_on_status AT %QD0.463 : UDINT;
      IM_SingleSignals_QF12_QF13_on_status AT %QD0.464 : UDINT;
      IM_SingleSignals_QF14_QF15_on_status AT %QD0.465 : UDINT;
      IM_SingleSignals_QF1_on_status AT %QD0.466 : UDINT;
      IM_SingleSignals_QF22_on_status AT %QD0.476 : UDINT;
      IM_SingleSignals_QF23_on_status AT %QD0.468 : UDINT;
      IM_SingleSignals_QF2_on_status AT %QD0.467 : UDINT;
      IM_SingleSignals_QF4_QF5_on_status AT %QD0.460 : UDINT;
      IM_SingleSignals_QF6_QF7_on_status AT %QD0.461 : UDINT;
      IM_SingleSignals_QF8_QF9_on_status AT %QD0.462 : UDINT;
      IM_SingleSignals_Vozb_AsinchHod_status AT %QD0.469 : UDINT;
      IM_SingleSignals_Vozb_ControlVozbuditela_status AT %QD0.470 : UDINT;
      IM_SingleSignals_Vozb_KontaktorON_status AT %QD0.471 : UDINT;
      IM_SingleSignals_Vozb_Overload_status AT %QD0.472 : UDINT;
      IM_SingleSignals_Vozb_ProboiVentila_status AT %QD0.473 : UDINT;
      IM_SingleSignals_Vozb_ReSynchronize_status AT %QD0.474 : UDINT;
      IM_SingleSignals_dP_gazgaz_Kran1_status AT %QD0.454 : UDINT;
      IM_SingleSignals_dP_oilgaz_low_status AT %QD0.475 : UDINT;
      IM_Ten_inCommand_ARM AT %QW0.447 : UINT;
      IM_Ten_status AT %QD0.448 : UDINT;
      IM_kran1_inCommand_ARM AT %QW0.427 : UINT;
      IM_kran1_status AT %QD0.428 : UDINT;
      IM_kran2_inCommand_ARM AT %QW0.429 : UINT;
      IM_kran2_status AT %QD0.430 : UDINT;
      IM_kran3b_inCommand_ARM AT %QW0.431 : UINT;
      IM_kran3b_status AT %QD0.432 : UDINT;
      IM_kran4_inCommand_ARM AT %QW0.433 : UINT;
      IM_kran4_status AT %QD0.434 : UDINT;
      IM_kran5_inCommand_ARM AT %QW0.435 : UINT;
      IM_kran5_status AT %QD0.436 : UDINT;
      IM_kran6_inCommand_ARM AT %QW0.437 : UINT;
      IM_kran6_status AT %QD0.438 : UDINT;
      IM_mv_inCommand_ARM AT %QW0.439 : UINT;
      IM_mv_status AT %QD0.440 : UDINT;
      IM_nu1_inCommand_ARM AT %QW0.441 : UINT;
      IM_nu1_status AT %QD0.442 : UDINT;
      IM_nu2_inCommand_ARM AT %QW0.443 : UINT;
      IM_nu2_status AT %QD0.444 : UDINT;
      IM_pns_inCommand_ARM AT %QW0.445 : UINT;
      IM_pns_status AT %QD0.446 : UDINT;
      IM_v1_Avom_inCommand_ARM AT %QW0.449 : UINT;
      IM_v1_Avom_status AT %QD0.450 : UDINT;
      IM_v2_Avom_inCommand_ARM AT %QW0.451 : UINT;
      IM_v2_Avom_status AT %QD0.452 : UDINT;
      algManager_Mode AT %QW0.732 : UINT;
      algoritms_AntiPompag_UgolVNA_Value AT %QL0.726 : LREAL;
      algoritms_AntiPompag_UgolVNA_inCommand_ARM AT %QW0.605 : UINT;
      algoritms_AntiPompag_UgolVNA_newValue AT %QL0.606 : LREAL;
      algoritms_AntiPompag_UgolVNA_status AT %QD0.725 : UDINT;
      algoritms_AntiPompag_q_Value AT %QL0.724 : LREAL;
      algoritms_AntiPompag_q_inCommand_ARM AT %QW0.604 : UINT;
      algoritms_AntiPompag_q_status AT %QD0.723 : UDINT;
      algoritms_AntiPompag_zapas_Value AT %QL0.728 : LREAL;
      algoritms_AntiPompag_zapas_inCommand_ARM AT %QW0.607 : UINT;
      algoritms_AntiPompag_zapas_status AT %QD0.727 : UDINT;
      algoritms_Apusk_Error AT %QD0.689 : UDINT;
      algoritms_Apusk_Start AT %QD0.688 : UDINT;
      algoritms_Apusk_Top AT %QD0.690 : UDINT;
      algoritms_Apusk_inCommand_ARM AT %QW0.555 : UINT;
      algoritms_Apusk_status AT %QD0.687 : UDINT;
      algoritms_AutoAvom_hysteresis_Value AT %QL0.716 : LREAL;
      algoritms_AutoAvom_hysteresis_inCommand_ARM AT %QW0.556 : UINT;
      algoritms_AutoAvom_hysteresis_newValue AT %QL0.557 : LREAL;
      algoritms_AutoAvom_hysteresis_status AT %QD0.715 : UDINT;
      algoritms_AutoAvom_inCommand_ARM AT %QW0.562 : UINT;
      algoritms_AutoAvom_on1Temperature_Value AT %QL0.712 : LREAL;
      algoritms_AutoAvom_on1Temperature_inCommand_ARM AT %QW0.558 : UINT;
      algoritms_AutoAvom_on1Temperature_newValue AT %QL0.559 : LREAL;
      algoritms_AutoAvom_on1Temperature_status AT %QD0.711 : UDINT;
      algoritms_AutoAvom_on2Temperature_Value AT %QL0.714 : LREAL;
      algoritms_AutoAvom_on2Temperature_inCommand_ARM AT %QW0.560 : UINT;
      algoritms_AutoAvom_on2Temperature_newValue AT %QL0.561 : LREAL;
      algoritms_AutoAvom_on2Temperature_status AT %QD0.713 : UDINT;
      algoritms_AutoAvom_status AT %QD0.710 : UDINT;
      algoritms_AutoPns_OffTimer AT %QW0.701 : UINT;
      algoritms_AutoPns_OnTimer AT %QW0.700 : UINT;
      algoritms_AutoPns_Ust_Run_Value AT %QL0.703 : LREAL;
      algoritms_AutoPns_Ust_Run_inCommand_ARM AT %QW0.567 : UINT;
      algoritms_AutoPns_Ust_Run_newValue AT %QL0.568 : LREAL;
      algoritms_AutoPns_Ust_Run_status AT %QD0.702 : UDINT;
      algoritms_AutoPns_Ust_Stop_Value AT %QL0.705 : LREAL;
      algoritms_AutoPns_Ust_Stop_inCommand_ARM AT %QW0.569 : UINT;
      algoritms_AutoPns_Ust_Stop_newValue AT %QL0.570 : LREAL;
      algoritms_AutoPns_Ust_Stop_status AT %QD0.704 : UDINT;
      algoritms_AutoPns_inCommand_ARM AT %QW0.571 : UINT;
      algoritms_AutoPns_status AT %QD0.699 : UDINT;
      algoritms_AutoTen_inCommand_ARM AT %QW0.610 : UINT;
      algoritms_AutoTen_offTemperature_Value AT %QL0.721 : LREAL;
      algoritms_AutoTen_offTemperature_inCommand_ARM AT %QW0.608 : UINT;
      algoritms_AutoTen_offTemperature_newValue AT %QL0.609 : LREAL;
      algoritms_AutoTen_offTemperature_status AT %QD0.720 : UDINT;
      algoritms_AutoTen_status AT %QD0.719 : UDINT;
      algoritms_Remont_inCommand_ARM AT %QW0.585 : UINT;
      algoritms_Remont_status AT %QD0.718 : UDINT;
      algoritms_RingToLine_Error AT %QD0.667 : UDINT;
      algoritms_RingToLine_Start AT %QD0.666 : UDINT;
      algoritms_RingToLine_Top AT %QD0.668 : UDINT;
      algoritms_RingToLine_inCommand_ARM AT %QW0.586 : UINT;
      algoritms_RingToLine_status AT %QD0.665 : UDINT;
      algoritms_SemiAutoPusk_Error AT %QD0.693 : UDINT;
      algoritms_SemiAutoPusk_Start AT %QD0.692 : UDINT;
      algoritms_SemiAutoPusk_Top AT %QD0.694 : UDINT;
      algoritms_SemiAutoPusk_cmdRun1ph_inCommand_ARM AT %QW0.587 : UINT;
      algoritms_SemiAutoPusk_cmdRun1ph_status AT %QD0.695 : UDINT;
      algoritms_SemiAutoPusk_cmdRun2ph_inCommand_ARM AT %QW0.588 : UINT;
      algoritms_SemiAutoPusk_cmdRun2ph_status AT %QD0.696 : UDINT;
      algoritms_SemiAutoPusk_cmdRun3ph_inCommand_ARM AT %QW0.589 : UINT;
      algoritms_SemiAutoPusk_cmdRun3ph_status AT %QD0.697 : UDINT;
      algoritms_SemiAutoPusk_cmdRun4ph_inCommand_ARM AT %QW0.590 : UINT;
      algoritms_SemiAutoPusk_cmdRun4ph_status AT %QD0.698 : UDINT;
      algoritms_SemiAutoPusk_inCommand_ARM AT %QW0.591 : UINT;
      algoritms_SemiAutoPusk_status AT %QD0.691 : UDINT;
      algoritms_TestProtection_inCommand_ARM AT %QW0.600 : UINT;
      algoritms_TestProtection_status AT %QD0.717 : UDINT;
      algoritms_ao_Error AT %QD0.617 : UDINT;
      algoritms_ao_Start AT %QD0.616 : UDINT;
      algoritms_ao_Top AT %QD0.618 : UDINT;
      algoritms_ao_inCommand_ARM AT %QW0.554 : UINT;
      algoritms_ao_status AT %QD0.619 : UDINT;
      algoritms_ao_waitKran_timer AT %QW0.620 : UINT;
      algoritms_autoNu_NotHasRezervNU AT %QX0.729 : BOOL;
      algoritms_autoNu_Ust_Swap_Value AT %QL0.708 : LREAL;
      algoritms_autoNu_Ust_Swap_inCommand_ARM AT %QW0.563 : UINT;
      algoritms_autoNu_Ust_Swap_newValue AT %QL0.564 : LREAL;
      algoritms_autoNu_Ust_Swap_status AT %QD0.707 : UDINT;
      algoritms_autoNu_inCommand_ARM AT %QW0.566 : UINT;
      algoritms_autoNu_mainNU_inCommand_ARM AT %QW0.565 : UINT;
      algoritms_autoNu_mainNU_status AT %QD0.722 : UDINT;
      algoritms_autoNu_status AT %QD0.706 : UDINT;
      algoritms_engineRun_BreakPuskTimer_timer AT %QW0.657 : UINT;
      algoritms_engineRun_Error AT %QD0.655 : UDINT;
      algoritms_engineRun_Start AT %QD0.654 : UDINT;
      algoritms_engineRun_Top AT %QD0.656 : UDINT;
      algoritms_engineRun_inCommand_ARM AT %QW0.572 : UINT;
      algoritms_engineRun_status AT %QD0.653 : UDINT;
      algoritms_filling_BreakPuskTimer_timer AT %QW0.662 : UINT;
      algoritms_filling_Error AT %QD0.660 : UDINT;
      algoritms_filling_Start AT %QD0.659 : UDINT;
      algoritms_filling_Top AT %QD0.661 : UDINT;
      algoritms_filling_inCommand_ARM AT %QW0.573 : UINT;
      algoritms_filling_status AT %QD0.658 : UDINT;
      algoritms_filling_waitAfterKran4_timer AT %QW0.663 : UINT;
      algoritms_filling_waitAfterKran5_timer AT %QW0.664 : UINT;
      algoritms_no_Error AT %QD0.612 : UDINT;
      algoritms_no_Start AT %QD0.611 : UDINT;
      algoritms_no_Top AT %QD0.613 : UDINT;
      algoritms_no_inCommand_ARM AT %QW0.574 : UINT;
      algoritms_no_status AT %QD0.614 : UDINT;
      algoritms_no_waitCloseKran_timer AT %QW0.615 : UINT;
      algoritms_ppu_Error AT %QD0.643 : UDINT;
      algoritms_ppu_Start AT %QD0.642 : UDINT;
      algoritms_ppu_Top AT %QD0.644 : UDINT;
      algoritms_ppu_inCommand_ARM AT %QW0.575 : UINT;
      algoritms_ppu_status AT %QD0.641 : UDINT;
      algoritms_puskK_Error AT %QD0.673 : UDINT;
      algoritms_puskK_Start AT %QD0.672 : UDINT;
      algoritms_puskK_Top AT %QD0.674 : UDINT;
      algoritms_puskK_inCommand_ARM AT %QW0.578 : UINT;
      algoritms_puskK_questionFilling_inCommand_ARM AT %QW0.576 : UINT;
      algoritms_puskK_questionFilling_status AT %QD0.677 : UDINT;
      algoritms_puskK_questionUnload_inCommand_ARM AT %QW0.577 : UINT;
      algoritms_puskK_questionUnload_status AT %QD0.678 : UDINT;
      algoritms_puskK_status AT %QD0.671 : UDINT;
      algoritms_puskK_wait720_timer AT %QW0.676 : UINT;
      algoritms_puskOilSystem_BreakPuskTimer_Poil_timer AT %QW0.649 : UINT;
      algoritms_puskOilSystem_BreakPuskTimer_dPmg_timer AT %QW0.650 : UINT;
      algoritms_puskOilSystem_Error AT %QD0.647 : UDINT;
      algoritms_puskOilSystem_Start AT %QD0.646 : UDINT;
      algoritms_puskOilSystem_Top AT %QD0.648 : UDINT;
      algoritms_puskOilSystem_Ust_dPmg_Value AT %QL0.652 : LREAL;
      algoritms_puskOilSystem_Ust_dPmg_inCommand_ARM AT %QW0.579 : UINT;
      algoritms_puskOilSystem_Ust_dPmg_newValue AT %QL0.580 : LREAL;
      algoritms_puskOilSystem_Ust_dPmg_status AT %QD0.651 : UDINT;
      algoritms_puskOilSystem_inCommand_ARM AT %QW0.581 : UINT;
      algoritms_puskOilSystem_status AT %QD0.645 : UDINT;
      algoritms_puskV_Error AT %QD0.681 : UDINT;
      algoritms_puskV_Start AT %QD0.680 : UDINT;
      algoritms_puskV_Top AT %QD0.682 : UDINT;
      algoritms_puskV_inCommand_ARM AT %QW0.584 : UINT;
      algoritms_puskV_questionFilling_inCommand_ARM AT %QW0.582 : UINT;
      algoritms_puskV_questionFilling_status AT %QD0.685 : UDINT;
      algoritms_puskV_questionMVoff_inCommand_ARM AT %QW0.583 : UINT;
      algoritms_puskV_questionMVoff_status AT %QD0.686 : UDINT;
      algoritms_puskV_status AT %QD0.679 : UDINT;
      algoritms_puskV_wait600_timer AT %QW0.684 : UINT;
      algoritms_testIm_TypeSwitch_inCommand_ARM AT %QW0.596 : UINT;
      algoritms_testIm_TypeSwitch_status AT %QD0.640 : UDINT;
      algoritms_testIm_inCommand_ARM AT %QW0.597 : UINT;
      algoritms_testIm_status AT %QD0.639 : UDINT;
      algoritms_testPms_BreakTest_timer AT %QW0.631 : UINT;
      algoritms_testPms_Error AT %QD0.628 : UDINT;
      algoritms_testPms_Start AT %QD0.627 : UDINT;
      algoritms_testPms_Top AT %QD0.629 : UDINT;
      algoritms_testPms_algContinue_inCommand_ARM AT %QW0.598 : UINT;
      algoritms_testPms_algContinue_status AT %QD0.669 : UDINT;
      algoritms_testPms_inCommand_ARM AT %QW0.599 : UINT;
      algoritms_testPms_status AT %QD0.630 : UDINT;
      algoritms_testdPmg_BreakTest_timer AT %QW0.636 : UINT;
      algoritms_testdPmg_Error AT %QD0.633 : UDINT;
      algoritms_testdPmg_Start AT %QD0.632 : UDINT;
      algoritms_testdPmg_Top AT %QD0.634 : UDINT;
      algoritms_testdPmg_Ust_dPLow_Value AT %QL0.638 : LREAL;
      algoritms_testdPmg_Ust_dPLow_inCommand_ARM AT %QW0.593 : UINT;
      algoritms_testdPmg_Ust_dPLow_newValue AT %QL0.594 : LREAL;
      algoritms_testdPmg_Ust_dPLow_status AT %QD0.637 : UDINT;
      algoritms_testdPmg_algContinue_inCommand_ARM AT %QW0.592 : UINT;
      algoritms_testdPmg_algContinue_status AT %QD0.670 : UDINT;
      algoritms_testdPmg_inCommand_ARM AT %QW0.595 : UINT;
      algoritms_testdPmg_status AT %QD0.635 : UDINT;
      algoritms_vibegPNS_Error AT %QD0.622 : UDINT;
      algoritms_vibegPNS_Start AT %QD0.621 : UDINT;
      algoritms_vibegPNS_Top AT %QD0.623 : UDINT;
      algoritms_vibegPNS_algContinue_inCommand_ARM AT %QW0.601 : UINT;
      algoritms_vibegPNS_algContinue_status AT %QD0.626 : UDINT;
      algoritms_vibegPNS_inCommand_ARM AT %QW0.602 : UINT;
      algoritms_vibegPNS_status AT %QD0.624 : UDINT;
      algoritms_vibegPNS_waitVibeg_timer AT %QW0.625 : UINT;
      protectManager_protectionInRemont AT %QX0.733 : BOOL;
      protections_AO_KC_inCommand_ARM AT %QW0.486 : UINT;
      protections_AO_KC_status AT %QD0.520 : UDINT;
      protections_AO_PRU_inCommand_ARM AT %QW0.487 : UINT;
      protections_AO_PRU_status AT %QD0.521 : UDINT;
      protections_AO_SHU_inCommand_ARM AT %QW0.488 : UINT;
      protections_AO_SHU_status AT %QD0.522 : UDINT;
      protections_BEAO_knSHU_inCommand_ARM AT %QW0.489 : UINT;
      protections_BEAO_knSHU_status AT %QD0.523 : UDINT;
      protections_DavlenieMaslaSmazkiDi_inCommand_ARM AT %QW0.490 : UINT;
      protections_DavlenieMaslaSmazkiDi_status AT %QD0.524 : UDINT;
      protections_EAO_PRU_inCommand_ARM AT %QW0.493 : UINT;
      protections_EAO_PRU_status AT %QD0.528 : UDINT;
      protections_Kran1sdvig_inCommand_ARM AT %QW0.517 : UINT;
      protections_Kran1sdvig_status AT %QD0.552 : UDINT;
      protections_Kran2sdvig_inCommand_ARM AT %QW0.518 : UINT;
      protections_Kran2sdvig_status AT %QD0.553 : UDINT;
      protections_Osevoi_sdvig_rotora_nagnetatelia_HA_inCommand_ARM AT %QW0.495 : UINT;
      protections_Osevoi_sdvig_rotora_nagnetatelia_HA_status AT %QD0.532 : UDINT;
      protections_OsevojSdvigLevyjDi_inCommand_ARM AT %QW0.496 : UINT;
      protections_OsevojSdvigLevyjDi_status AT %QD0.530 : UDINT;
      protections_OsevojSdvigPravyjDi_inCommand_ARM AT %QW0.497 : UINT;
      protections_OsevojSdvigPravyjDi_status AT %QD0.531 : UDINT;
      protections_P_masla_smazki_nizkoe_LA_inCommand_ARM AT %QW0.519 : UINT;
      protections_P_masla_smazki_nizkoe_LA_status AT %QD0.525 : UDINT;
      protections_Srab_BEAO_inCommand_ARM AT %QW0.498 : UINT;
      protections_Srab_BEAO_status AT %QD0.534 : UDINT;
      protections_T_gaza_na_vykhode_nagnetatelia_HA_inCommand_ARM AT %QW0.499 : UINT;
      protections_T_gaza_na_vykhode_nagnetatelia_HA_status AT %QD0.533 : UDINT;
      protections_T_opornogo_podshipnika_nagnetatelia_t1_HA_inCommand_ARM AT %QW0.500 : UINT;
      protections_T_opornogo_podshipnika_nagnetatelia_t1_HA_status AT %QD0.535 : UDINT;
      protections_T_opornogo_podshipnika_nagnetatelia_t2_HA_inCommand_ARM AT %QW0.501 : UINT;
      protections_T_opornogo_podshipnika_nagnetatelia_t2_HA_status AT %QD0.536 : UDINT;
      protections_T_opornogo_podshipnika_nagnetatelia_t3_HA_inCommand_ARM AT %QW0.502 : UINT;
      protections_T_opornogo_podshipnika_nagnetatelia_t3_HA_status AT %QD0.537 : UDINT;
      protections_T_opornoupornogo_podshipnika_nagnetatelia_t4_HA_inCommand_ARM AT %QW0.503 : UINT;
      protections_T_opornoupornogo_podshipnika_nagnetatelia_t4_HA_status AT %QD0.538 : UDINT;
      protections_T_perednego_opornogo_podshipnika_dvigatelia_t1_HA_inCommand_ARM AT %QW0.504 : UINT;
      protections_T_perednego_opornogo_podshipnika_dvigatelia_t1_HA_status AT %QD0.539 : UDINT;
      protections_T_podshipnika_reduktora_t1_HA_inCommand_ARM AT %QW0.505 : UINT;
      protections_T_podshipnika_reduktora_t1_HA_status AT %QD0.541 : UDINT;
      protections_T_podshipnika_reduktora_t2_HA_inCommand_ARM AT %QW0.506 : UINT;
      protections_T_podshipnika_reduktora_t2_HA_status AT %QD0.542 : UDINT;
      protections_T_podshipnika_reduktora_t3_HA_inCommand_ARM AT %QW0.507 : UINT;
      protections_T_podshipnika_reduktora_t3_HA_status AT %QD0.543 : UDINT;
      protections_T_podshipnika_reduktora_t4_HA_inCommand_ARM AT %QW0.508 : UINT;
      protections_T_podshipnika_reduktora_t4_HA_status AT %QD0.544 : UDINT;
      protections_T_zadnego_opornogo_podshipnika_dvigatelia_t2_HA_inCommand_ARM AT %QW0.509 : UINT;
      protections_T_zadnego_opornogo_podshipnika_dvigatelia_t2_HA_status AT %QD0.540 : UDINT;
      protections_Uroven_masla_v_maslobake_LA_inCommand_ARM AT %QW0.510 : UINT;
      protections_Uroven_masla_v_maslobake_LA_status AT %QD0.545 : UDINT;
      protections_Vibratciia_STD_t1_HA_inCommand_ARM AT %QW0.515 : UINT;
      protections_Vibratciia_STD_t1_HA_status AT %QD0.550 : UDINT;
      protections_Vibratciia_STD_t2_HA_inCommand_ARM AT %QW0.516 : UINT;
      protections_Vibratciia_STD_t2_HA_status AT %QD0.551 : UDINT;
      protections_Vibratciia_rotora_nagnetatelia_t1_HA_inCommand_ARM AT %QW0.511 : UINT;
      protections_Vibratciia_rotora_nagnetatelia_t1_HA_status AT %QD0.546 : UDINT;
      protections_Vibratciia_rotora_nagnetatelia_t2_HA_inCommand_ARM AT %QW0.512 : UINT;
      protections_Vibratciia_rotora_nagnetatelia_t2_HA_status AT %QD0.547 : UDINT;
      protections_Vibratciia_rotora_nagnetatelia_t3_HA_inCommand_ARM AT %QW0.513 : UINT;
      protections_Vibratciia_rotora_nagnetatelia_t3_HA_status AT %QD0.548 : UDINT;
      protections_Vibratciia_rotora_nagnetatelia_t4_HA_inCommand_ARM AT %QW0.514 : UINT;
      protections_Vibratciia_rotora_nagnetatelia_t4_HA_status AT %QD0.549 : UDINT;
      protections_dP_masloGaz_LowDI_inCommand_ARM AT %QW0.492 : UINT;
      protections_dP_masloGaz_LowDI_status AT %QD0.527 : UDINT;
      protections_dP_maslogaz_LA_inCommand_ARM AT %QW0.491 : UINT;
      protections_dP_maslogaz_LA_status AT %QD0.526 : UDINT;
      protections_mvOff_inCommand_ARM AT %QW0.494 : UINT;
      protections_mvOff_status AT %QD0.529 : UDINT;
      algoritms_autoNu_Reset_HasNU AT %QX0.731 : BOOL;
      A1_10_err_mode AT %QW0.825 : UINT;
      A1_11_err_mode AT %QW0.826 : UINT;
      A1_12_err_mode AT %QW0.827 : UINT;
      A1_13_err_mode AT %QW0.828 : UINT;
      A1_14_err_mode AT %QW0.829 : UINT;
      A1_15_err_mode AT %QW0.830 : UINT;
      A1_1_err_mode AT %QW0.816 : UINT;
      A1_2_err_mode AT %QW0.817 : UINT;
      A1_3_err_mode AT %QW0.818 : UINT;
      A1_4_err_mode AT %QW0.819 : UINT;
      A1_5_err_mode AT %QW0.820 : UINT;
      A1_6_err_mode AT %QW0.821 : UINT;
      A1_7_err_mode AT %QW0.822 : UINT;
      A1_8_err_mode AT %QW0.823 : UINT;
      A1_9_err_mode AT %QW0.824 : UINT;
      A2_10_err_mode AT %QW0.840 : UINT;
      A2_11_err_mode AT %QW0.841 : UINT;
      A2_12_err_mode AT %QW0.842 : UINT;
      A2_13_err_mode AT %QW0.843 : UINT;
      A2_14_err_mode AT %QW0.844 : UINT;
      A2_15_err_mode AT %QW0.845 : UINT;
      A2_1_err_mode AT %QW0.831 : UINT;
      A2_2_err_mode AT %QW0.832 : UINT;
      A2_3_err_mode AT %QW0.833 : UINT;
      A2_4_err_mode AT %QW0.834 : UINT;
      A2_5_err_mode AT %QW0.835 : UINT;
      A2_6_err_mode AT %QW0.836 : UINT;
      A2_7_err_mode AT %QW0.837 : UINT;
      A2_8_err_mode AT %QW0.838 : UINT;
      A2_9_err_mode AT %QW0.839 : UINT;
      AI_0_dblValue AT %QL0.736 : LREAL;
      AI_10_dblValue AT %QL0.746 : LREAL;
      AI_11_dblValue AT %QL0.747 : LREAL;
      AI_12_dblValue AT %QL0.748 : LREAL;
      AI_13_dblValue AT %QL0.749 : LREAL;
      AI_14_dblValue AT %QL0.750 : LREAL;
      AI_15_dblValue AT %QL0.751 : LREAL;
      AI_16_dblValue AT %QL0.752 : LREAL;
      AI_17_dblValue AT %QL0.753 : LREAL;
      AI_18_dblValue AT %QL0.754 : LREAL;
      AI_19_dblValue AT %QL0.755 : LREAL;
      AI_1_dblValue AT %QL0.737 : LREAL;
      AI_20_dblValue AT %QL0.756 : LREAL;
      AI_21_dblValue AT %QL0.757 : LREAL;
      AI_22_dblValue AT %QL0.758 : LREAL;
      AI_23_dblValue AT %QL0.759 : LREAL;
      AI_24_dblValue AT %QL0.760 : LREAL;
      AI_25_dblValue AT %QL0.761 : LREAL;
      AI_26_dblValue AT %QL0.762 : LREAL;
      AI_27_dblValue AT %QL0.763 : LREAL;
      AI_28_dblValue AT %QL0.764 : LREAL;
      AI_29_dblValue AT %QL0.765 : LREAL;
      AI_2_dblValue AT %QL0.738 : LREAL;
      AI_30_dblValue AT %QL0.766 : LREAL;
      AI_31_dblValue AT %QL0.767 : LREAL;
      AI_32_dblValue AT %QL0.768 : LREAL;
      AI_33_dblValue AT %QL0.769 : LREAL;
      AI_34_dblValue AT %QL0.770 : LREAL;
      AI_35_dblValue AT %QL0.771 : LREAL;
      AI_36_dblValue AT %QL0.772 : LREAL;
      AI_37_dblValue AT %QL0.773 : LREAL;
      AI_38_dblValue AT %QL0.774 : LREAL;
      AI_39_dblValue AT %QL0.775 : LREAL;
      AI_3_dblValue AT %QL0.739 : LREAL;
      AI_40_dblValue AT %QL0.776 : LREAL;
      AI_41_dblValue AT %QL0.777 : LREAL;
      AI_42_dblValue AT %QL0.778 : LREAL;
      AI_43_dblValue AT %QL0.779 : LREAL;
      AI_44_dblValue AT %QL0.780 : LREAL;
      AI_45_dblValue AT %QL0.781 : LREAL;
      AI_46_dblValue AT %QL0.782 : LREAL;
      AI_47_dblValue AT %QL0.783 : LREAL;
      AI_48_dblValue AT %QL0.784 : LREAL;
      AI_49_dblValue AT %QL0.785 : LREAL;
      AI_4_dblValue AT %QL0.740 : LREAL;
      AI_50_dblValue AT %QL0.786 : LREAL;
      AI_51_dblValue AT %QL0.787 : LREAL;
      AI_52_dblValue AT %QL0.788 : LREAL;
      AI_53_dblValue AT %QL0.789 : LREAL;
      AI_54_dblValue AT %QL0.790 : LREAL;
      AI_55_dblValue AT %QL0.791 : LREAL;
      AI_56_dblValue AT %QL0.792 : LREAL;
      AI_57_dblValue AT %QL0.793 : LREAL;
      AI_58_dblValue AT %QL0.794 : LREAL;
      AI_59_dblValue AT %QL0.795 : LREAL;
      AI_5_dblValue AT %QL0.741 : LREAL;
      AI_60_dblValue AT %QL0.796 : LREAL;
      AI_61_dblValue AT %QL0.797 : LREAL;
      AI_62_dblValue AT %QL0.798 : LREAL;
      AI_63_dblValue AT %QL0.799 : LREAL;
      AI_64_dblValue AT %QL0.800 : LREAL;
      AI_65_dblValue AT %QL0.801 : LREAL;
      AI_66_dblValue AT %QL0.802 : LREAL;
      AI_67_dblValue AT %QL0.803 : LREAL;
      AI_68_dblValue AT %QL0.804 : LREAL;
      AI_69_dblValue AT %QL0.805 : LREAL;
      AI_6_dblValue AT %QL0.742 : LREAL;
      AI_70_dblValue AT %QL0.806 : LREAL;
      AI_71_dblValue AT %QL0.807 : LREAL;
      AI_72_dblValue AT %QL0.808 : LREAL;
      AI_73_dblValue AT %QL0.809 : LREAL;
      AI_74_dblValue AT %QL0.810 : LREAL;
      AI_75_dblValue AT %QL0.811 : LREAL;
      AI_76_dblValue AT %QL0.812 : LREAL;
      AI_77_dblValue AT %QL0.813 : LREAL;
      AI_78_dblValue AT %QL0.814 : LREAL;
      AI_79_dblValue AT %QL0.815 : LREAL;
      AI_7_dblValue AT %QL0.743 : LREAL;
      AI_8_dblValue AT %QL0.744 : LREAL;
      AI_9_dblValue AT %QL0.745 : LREAL;
      BS_Core1 AT %QD0.603 : REAL;
      BS_Core2 AT %QD0.675 : REAL;
      BS_Core3 AT %QD0.683 : REAL;
      BS_Core4 AT %QD0.709 : REAL;
      BS_FreeMemory AT %QD0.730 : REAL;
      BS_Temp1 AT %QD0.734 : REAL;
      BS_Temp2 AT %QD0.735 : REAL;
      DI_0_1_wValue AT %QD0.852 : UDINT;
      DI_10_11_wValue AT %QD0.857 : UDINT;
      DI_12_13_wValue AT %QD0.858 : UDINT;
      DI_14_15_wValue AT %QD0.859 : UDINT;
      DI_16_17_wValue AT %QD0.860 : UDINT;
      DI_18_19_wValue AT %QD0.861 : UDINT;
      DI_20_21_wValue AT %QD0.862 : UDINT;
      DI_2_3_wValue AT %QD0.853 : UDINT;
      DI_4_5_wValue AT %QD0.854 : UDINT;
      DI_6_7_wValue AT %QD0.855 : UDINT;
      DI_8_9_wValue AT %QD0.856 : UDINT;
      DO_0_wValue AT %QW0.846 : UINT;
      DO_1_wValue AT %QW0.847 : UINT;
      DO_2_wValue AT %QW0.848 : UINT;
      DO_3_wValue AT %QW0.849 : UINT;
      DO_4_wValue AT %QW0.850 : UINT;
      DO_5_wValue AT %QW0.851 : UINT;
      AI_T_vnytri_shkafa_HL AT %QL0.866 : LREAL;
      AI_T_vnytri_shkafa_HW AT %QL0.870 : LREAL;
      AI_T_vnytri_shkafa_LL AT %QL0.867 : LREAL;
      AI_T_vnytri_shkafa_LW AT %QL0.872 : LREAL;
      AI_T_vnytri_shkafa_command AT %QW0.863 : UINT;
      AI_T_vnytri_shkafa_newHL AT %QL0.868 : LREAL;
      AI_T_vnytri_shkafa_newHW AT %QL0.871 : LREAL;
      AI_T_vnytri_shkafa_newLL AT %QL0.869 : LREAL;
      AI_T_vnytri_shkafa_newLW AT %QL0.873 : LREAL;
      AI_T_vnytri_shkafa_status AT %QD0.864 : UDINT;
      AI_T_vnytri_shkafa_value AT %QL0.865 : LREAL;
      AI_dPmaslo_gaz_MaxChangeDown AT %QL0.877 : LREAL;
      AI_dPmaslo_gaz_MaxChangeUP AT %QL0.876 : LREAL;
      AI_dPmaslo_gaz_newMaxChangeDown AT %QL0.875 : LREAL;
      AI_dPmaslo_gaz_newMaxChangeUP AT %QL0.874 : LREAL;
    END_VAR
    TASK task0(INTERVAL := T#20ms,PRIORITY := 0);
    PROGRAM instance0 WITH task0 : program0;
  END_RESOURCE
END_CONFIGURATION
